C03645=1176.042,92.652,-51.203,-179.040,6.178,148.830
C03646=1176.047,92.403,-51.185,-179.044,6.176,148.831
C03647=1176.052,92.154,-51.167,-179.046,6.175,148.831
C03648=1176.057,91.904,-51.149,-179.048,6.174,148.832
C03649=1176.062,91.655,-51.131,-179.051,6.173,148.832
C03650=1176.066,91.406,-51.113,-179.054,6.172,148.833
C03651=1176.071,91.156,-51.095,-179.056,6.171,148.833
C03652=1176.076,90.906,-51.077,-179.059,6.169,148.834
C03653=1176.081,90.657,-51.059,-179.061,6.168,148.834
C03654=1176.086,90.408,-51.042,-179.064,6.167,148.835
C03655=1176.091,90.159,-51.024,-179.067,6.166,148.835
C03656=1176.096,89.910,-51.006,-179.070,6.165,148.836
C03657=1176.101,89.660,-50.988,-179.073,6.163,148.836
C03658=1176.106,89.411,-50.970,-179.075,6.162,148.837
C03659=1176.111,89.162,-50.952,-179.078,6.161,148.837
C03660=1176.116,88.912,-50.934,-179.080,6.160,148.838
C03661=1176.120,88.664,-50.917,-179.083,6.159,148.839
C03662=1176.125,88.414,-50.900,-179.085,6.158,148.839
C03663=1176.130,88.165,-50.882,-179.089,6.156,148.840
C03664=1176.135,87.915,-50.864,-179.091,6.155,148.840
C03665=1176.140,87.666,-50.846,-179.093,6.154,148.840
C03666=1176.145,87.416,-50.828,-179.096,6.153,148.841
C03667=1176.150,87.167,-50.811,-179.099,6.151,148.842
C03668=1176.155,86.918,-50.793,-179.101,6.151,148.842
C03669=1176.159,86.669,-50.776,-179.104,6.149,148.843
C03670=1176.164,86.419,-50.758,-179.106,6.148,148.843
C03671=1176.169,86.170,-50.740,-179.109,6.147,148.844
C03672=1176.174,85.920,-50.723,-179.112,6.146,148.844
C03673=1176.179,85.671,-50.705,-179.115,6.145,148.845
C03674=1176.184,85.422,-50.687,-179.117,6.144,148.845
C03675=1176.189,85.173,-50.670,-179.120,6.142,148.846
C03676=1176.193,84.923,-50.652,-179.122,6.142,148.846
C03677=1176.198,84.674,-50.634,-179.125,6.140,148.847
C03678=1176.204,84.424,-50.617,-179.128,6.139,148.847
C03679=1176.209,84.175,-50.599,-179.130,6.138,148.848
C03680=1176.213,83.926,-50.582,-179.133,6.137,148.848
C03681=1176.218,83.677,-50.564,-179.136,6.135,148.849
C03682=1176.223,83.427,-50.547,-179.138,6.135,148.849
C03683=1176.228,83.178,-50.529,-179.141,6.133,148.850
C03684=1176.232,82.929,-50.512,-179.144,6.133,148.851
C03685=1176.237,82.679,-50.494,-179.146,6.131,148.851
C03686=1176.242,82.430,-50.476,-179.149,6.130,148.852
C03687=1176.248,82.180,-50.459,-179.152,6.129,148.852
C03688=1176.252,81.931,-50.442,-179.154,6.128,148.852
C03689=1176.257,81.681,-50.424,-179.157,6.126,148.853
C03690=1176.262,81.432,-50.406,-179.159,6.125,148.854
C03691=1176.267,81.183,-50.390,-179.162,6.124,148.854
C03692=1176.272,80.934,-50.372,-179.165,6.123,148.855
C03693=1176.277,80.665,-50.353,-179.168,6.122,148.855
C03694=1176.283,80.397,-50.335,-179.170,6.121,148.856
C03695=1176.288,80.129,-50.316,-179.173,6.120,148.856
C03696=1176.293,79.860,-50.298,-179.176,6.118,148.857
C03697=1176.298,79.611,-50.280,-179.179,6.117,148.857
C03698=1176.303,79.361,-50.262,-179.182,6.116,148.858
C03699=1176.308,79.112,-50.246,-179.184,6.115,148.858
C03700=1176.312,78.863,-50.228,-179.187,6.114,148.859
C03701=1176.317,78.613,-50.211,-179.189,6.113,148.860
C03702=1176.323,78.364,-50.194,-179.192,6.112,148.860
C03703=1176.328,78.115,-50.176,-179.195,6.111,148.861
C03704=1176.332,77.866,-50.159,-179.197,6.110,148.861
C03705=1176.337,77.616,-50.142,-179.200,6.108,148.862
C03706=1176.342,77.367,-50.124,-179.202,6.108,148.862
C03707=1176.347,77.117,-50.108,-179.205,6.106,148.863
C03708=1176.353,76.868,-50.091,-179.207,6.105,148.863
C03709=1176.357,76.619,-50.073,-179.211,6.104,148.864
C03710=1176.362,76.369,-50.056,-179.213,6.103,148.864
C03711=1176.366,76.120,-50.039,-179.216,6.102,148.865
C03712=1176.372,75.870,-50.022,-179.218,6.101,148.865
C03713=1176.377,75.621,-50.004,-179.221,6.100,148.866
C03714=1176.382,75.372,-49.988,-179.223,6.099,148.866
C03715=1176.387,75.122,-49.971,-179.226,6.098,148.867
C03716=1176.391,74.873,-49.954,-179.229,6.096,148.868
C03717=1176.396,74.624,-49.936,-179.231,6.096,148.868
C03718=1176.401,74.374,-49.919,-179.234,6.094,148.869
C03719=1176.407,74.125,-49.902,-179.237,6.094,148.869
C03720=1176.411,73.876,-49.886,-179.239,6.093,148.870
C03721=1176.416,73.626,-49.868,-179.242,6.091,148.870
C03722=1176.420,73.377,-49.851,-179.244,6.091,148.871
C03723=1176.426,73.127,-49.834,-179.248,6.089,148.871
C03724=1176.431,72.878,-49.817,-179.250,6.088,148.872
C03725=1176.436,72.629,-49.800,-179.253,6.087,148.873
C03726=1176.440,72.379,-49.783,-179.255,6.086,148.873
C03727=1176.446,72.129,-49.766,-179.258,6.086,148.874
C03728=1176.451,71.880,-49.750,-179.260,6.084,148.874
C03729=1176.455,71.632,-49.733,-179.263,6.083,148.875
C03730=1176.460,71.382,-49.715,-179.266,6.082,148.875
C03731=1176.465,71.132,-49.699,-179.268,6.081,148.876
C03732=1176.470,70.883,-49.682,-179.271,6.080,148.876
C03733=1176.475,70.634,-49.665,-179.273,6.079,148.877
C03734=1176.480,70.384,-49.648,-179.276,6.078,148.877
C03735=1176.485,70.135,-49.631,-179.279,6.076,148.878
C03736=1176.490,69.886,-49.615,-179.281,6.076,148.878
C03737=1176.495,69.636,-49.598,-179.284,6.074,148.879
C03738=1176.499,69.386,-49.581,-179.287,6.074,148.880
C03739=1176.505,69.137,-49.564,-179.289,6.073,148.880
C03740=1176.510,68.888,-49.547,-179.292,6.071,148.881
C03741=1176.514,68.638,-49.531,-179.294,6.070,148.881
C03742=1176.520,68.389,-49.514,-179.297,6.069,148.882
C03743=1176.524,68.140,-49.497,-179.300,6.069,148.882
C03744=1176.529,67.890,-49.480,-179.302,6.068,148.883
C03745=1176.535,67.641,-49.463,-179.305,6.066,148.883
C03746=1176.539,67.392,-49.447,-179.307,6.066,148.884
C03747=1176.544,67.142,-49.430,-179.310,6.065,148.885
C03748=1176.549,66.892,-49.413,-179.313,6.063,148.885
C03749=1176.554,66.644,-49.397,-179.315,6.063,148.886
C03750=1176.559,66.394,-49.380,-179.318,6.061,148.886
C03751=1176.564,66.145,-49.363,-179.321,6.061,148.887
C03752=1176.569,65.896,-49.346,-179.323,6.060,148.887
C03753=1176.574,65.645,-49.330,-179.326,6.058,148.888
C03754=1176.579,65.397,-49.314,-179.328,6.057,148.888
C03755=1176.584,65.147,-49.297,-179.331,6.057,148.889
C03756=1176.588,64.897,-49.280,-179.334,6.055,148.889
C03757=1176.593,64.649,-49.264,-179.336,6.055,148.890
C03758=1176.599,64.399,-49.247,-179.339,6.053,148.890
C03759=1176.603,64.149,-49.230,-179.342,6.053,148.891
C03760=1176.609,63.900,-49.214,-179.344,6.052,148.892
C03761=1176.613,63.650,-49.198,-179.347,6.050,148.892
C03762=1176.619,63.401,-49.181,-179.349,6.049,148.893
C03763=1176.623,63.152,-49.164,-179.352,6.049,148.893
C03764=1176.628,62.902,-49.147,-179.355,6.047,148.894
C03765=1176.633,62.653,-49.132,-179.357,6.047,148.894
C03766=1176.638,62.404,-49.115,-179.359,6.046,148.895
C03767=1176.644,62.154,-49.098,-179.363,6.045,148.895
C03768=1176.648,61.905,-49.082,-179.365,6.044,148.896
C03769=1176.653,61.655,-49.066,-179.368,6.042,148.897
C03770=1176.658,61.406,-49.049,-179.371,6.042,148.897
C03771=1176.662,61.157,-49.033,-179.373,6.041,148.898
C03772=1176.668,60.907,-49.017,-179.376,6.040,148.898
C03773=1176.673,60.657,-49.000,-179.378,6.039,148.899
C03774=1176.678,60.409,-48.984,-179.381,6.038,148.899
C03775=1176.683,60.158,-48.968,-179.383,6.036,148.900
C03776=1176.688,59.910,-48.951,-179.386,6.036,148.901
C03777=1176.692,59.660,-48.935,-179.388,6.035,148.901
C03778=1176.697,59.410,-48.919,-179.391,6.034,148.902
C03779=1176.702,59.161,-48.902,-179.394,6.033,148.902
C03780=1176.707,58.912,-48.885,-179.396,6.032,148.903
C03781=1176.713,58.662,-48.869,-179.399,6.031,148.903
C03782=1176.717,58.413,-48.853,-179.402,6.030,148.904
C03783=1176.722,58.164,-48.837,-179.404,6.030,148.905
C03784=1176.727,57.914,-48.821,-179.407,6.028,148.905
C03785=1176.732,57.665,-48.804,-179.410,6.027,148.906
C03786=1176.737,57.415,-48.788,-179.412,6.027,148.906
C03787=1176.742,57.166,-48.772,-179.415,6.025,148.907
C03788=1176.747,56.916,-48.756,-179.417,6.024,148.907
C03789=1176.752,56.667,-48.740,-179.420,6.024,148.908
C03790=1176.756,56.418,-48.723,-179.423,6.022,148.908
C03791=1176.762,56.168,-48.707,-179.425,6.022,148.909
C03792=1176.767,55.919,-48.690,-179.427,6.021,148.909
C03793=1176.772,55.669,-48.675,-179.431,6.019,148.910
C03794=1176.777,55.420,-48.658,-179.433,6.019,148.911
C03795=1176.782,55.170,-48.642,-179.435,6.018,148.911
C03796=1176.787,54.921,-48.626,-179.438,6.018,148.912
C03797=1176.792,54.652,-48.609,-179.441,6.016,148.912
C03798=1176.798,54.384,-48.592,-179.443,6.015,148.913
C03799=1176.803,54.115,-48.575,-179.447,6.014,148.914
C03800=1176.808,53.846,-48.557,-179.449,6.014,148.914
C03801=1176.814,53.597,-48.541,-179.452,6.012,148.915
C03802=1176.819,53.348,-48.525,-179.455,6.011,148.915
C03803=1176.823,53.098,-48.509,-179.457,6.010,148.916
C03804=1176.829,52.849,-48.493,-179.460,6.009,148.916
C03805=1176.833,52.600,-48.476,-179.462,6.008,148.917
C03806=1176.839,52.350,-48.461,-179.465,6.008,148.918
C03807=1176.843,52.100,-48.445,-179.468,6.006,148.918
C03808=1176.849,51.851,-48.429,-179.470,6.006,148.919
C03809=1176.853,51.602,-48.414,-179.473,6.005,148.919
C03810=1176.858,51.352,-48.398,-179.475,6.004,148.920
C03811=1176.863,51.103,-48.381,-179.478,6.003,148.920
C03812=1176.868,50.853,-48.365,-179.480,6.002,148.921
C03813=1176.873,50.604,-48.350,-179.483,6.001,148.922
C03814=1176.878,50.355,-48.334,-179.486,6.000,148.922
C03815=1176.883,50.105,-48.318,-179.488,5.999,148.923
C03816=1176.888,49.856,-48.302,-179.491,5.999,148.923
C03817=1176.894,49.607,-48.286,-179.493,5.998,148.924
C03818=1176.898,49.357,-48.270,-179.496,5.997,148.924
C03819=1176.903,49.108,-48.255,-179.498,5.996,148.925
C03820=1176.908,48.857,-48.239,-179.501,5.995,148.926
C03821=1176.913,48.609,-48.222,-179.504,5.995,148.926
C03822=1176.918,48.359,-48.207,-179.506,5.993,148.927
C03823=1176.923,48.109,-48.191,-179.509,5.993,148.927
C03824=1176.928,47.860,-48.175,-179.511,5.992,148.928
C03825=1176.933,47.611,-48.160,-179.515,5.990,148.928
C03826=1176.938,47.361,-48.144,-179.517,5.989,148.929
C03827=1176.943,47.112,-48.128,-179.519,5.989,148.930
C03828=1176.948,46.862,-48.112,-179.522,5.988,148.930
C03829=1176.953,46.612,-48.097,-179.525,5.987,148.931
C03830=1176.957,46.364,-48.081,-179.527,5.986,148.931
C03831=1176.963,46.114,-48.065,-179.529,5.985,148.932
C03832=1176.968,45.864,-48.049,-179.532,5.985,148.932
C03833=1176.973,45.615,-48.034,-179.535,5.984,148.933
C03834=1176.978,45.366,-48.019,-179.537,5.983,148.934
C03835=1176.982,45.116,-48.003,-179.540,5.982,148.934
C03836=1176.988,44.866,-47.987,-179.542,5.981,148.935
C03837=1176.993,44.618,-47.971,-179.546,5.980,148.935
C03838=1176.998,44.368,-47.955,-179.548,5.979,148.936
C03839=1177.002,44.118,-47.940,-179.550,5.979,148.936
C03840=1177.008,43.869,-47.924,-179.553,5.978,148.937
C03841=1177.013,43.619,-47.909,-179.556,5.976,148.938
C03842=1177.017,43.370,-47.893,-179.558,5.976,148.938
C03843=1177.023,43.120,-47.878,-179.560,5.975,148.939
C03844=1177.028,42.871,-47.862,-179.563,5.975,148.939
C03845=1177.033,42.621,-47.847,-179.566,5.973,148.940
C03846=1177.037,42.372,-47.831,-179.569,5.972,148.940
C03847=1177.043,42.122,-47.816,-179.571,5.972,148.941
C03848=1177.048,41.873,-47.800,-179.573,5.971,148.942
C03849=1177.053,41.624,-47.785,-179.576,5.971,148.942
C03850=1177.058,41.374,-47.769,-179.579,5.969,148.943
C03851=1177.063,41.124,-47.754,-179.581,5.968,148.943
C03852=1177.068,40.875,-47.739,-179.584,5.968,148.944
C03853=1177.073,40.626,-47.723,-179.586,5.967,148.945
C03854=1177.078,40.376,-47.707,-179.589,5.966,148.945
C03855=1177.082,40.127,-47.692,-179.592,5.965,148.946
C03856=1177.088,39.877,-47.676,-179.594,5.964,148.946
C03857=1177.093,39.628,-47.661,-179.597,5.964,148.947
C03858=1177.098,39.379,-47.646,-179.599,5.963,148.947
C03859=1177.103,39.129,-47.630,-179.602,5.962,148.948
C03860=1177.107,38.880,-47.615,-179.605,5.961,148.949
C03861=1177.113,38.629,-47.600,-179.607,5.960,148.949
C03862=1177.118,38.380,-47.584,-179.610,5.960,148.950
C03863=1177.123,38.131,-47.569,-179.612,5.958,148.950
C03864=1177.128,37.882,-47.554,-179.615,5.958,148.951
C03865=1177.132,37.632,-47.539,-179.618,5.957,148.952
C03866=1177.138,37.382,-47.523,-179.620,5.956,148.952
C03867=1177.143,37.133,-47.507,-179.622,5.956,148.953
C03868=1177.148,36.883,-47.493,-179.625,5.954,148.953
C03869=1177.154,36.634,-47.477,-179.628,5.954,148.954
C03870=1177.158,36.385,-47.462,-179.630,5.953,148.955
C03871=1177.164,36.135,-47.447,-179.633,5.952,148.955
C03872=1177.168,35.886,-47.432,-179.635,5.952,148.956
C03873=1177.173,35.636,-47.417,-179.638,5.950,148.956
C03874=1177.178,35.386,-47.402,-179.641,5.950,148.957
C03875=1177.183,35.137,-47.386,-179.643,5.949,148.958
C03876=1177.188,34.888,-47.371,-179.645,5.948,148.958
C03877=1177.193,34.639,-47.356,-179.648,5.948,148.959
C03878=1177.198,34.389,-47.341,-179.651,5.946,148.959
C03879=1177.204,34.139,-47.326,-179.653,5.946,148.960
C03880=1177.208,33.890,-47.310,-179.656,5.945,148.960
C03881=1177.213,33.640,-47.295,-179.658,5.944,148.961
C03882=1177.218,33.391,-47.280,-179.661,5.944,148.962
C03883=1177.224,33.141,-47.265,-179.664,5.943,148.962
C03884=1177.228,32.892,-47.250,-179.666,5.942,148.963
C03885=1177.234,32.642,-47.235,-179.669,5.941,148.963
C03886=1177.239,32.393,-47.220,-179.671,5.940,148.964
C03887=1177.244,32.144,-47.204,-179.674,5.940,148.964
C03888=1177.249,31.894,-47.190,-179.676,5.939,148.965
C03889=1177.254,31.645,-47.175,-179.679,5.938,148.966
C03890=1177.259,31.394,-47.160,-179.682,5.937,148.966
C03891=1177.263,31.145,-47.145,-179.684,5.937,148.967
C03892=1177.269,30.896,-47.129,-179.687,5.936,148.967
C03893=1177.274,30.646,-47.115,-179.689,5.935,148.968
C03894=1177.278,30.397,-47.100,-179.691,5.934,148.969
C03895=1177.284,30.147,-47.084,-179.695,5.933,148.969
C03896=1177.289,29.898,-47.070,-179.697,5.933,148.970
C03897=1177.294,29.648,-47.055,-179.699,5.932,148.970
C03898=1177.299,29.399,-47.040,-179.702,5.931,148.971
C03899=1177.304,29.149,-47.025,-179.705,5.931,148.972
C03900=1177.309,28.899,-47.010,-179.707,5.930,148.972
C03901=1177.314,28.631,-46.995,-179.710,5.929,148.973
C03902=1177.320,28.362,-46.978,-179.713,5.928,148.973
C03903=1177.325,28.093,-46.962,-179.715,5.928,148.974
C03904=1177.330,27.825,-46.946,-179.718,5.926,148.975
C03905=1177.336,27.575,-46.931,-179.721,5.925,148.975
C03906=1177.341,27.325,-46.916,-179.723,5.925,148.976
C03907=1177.345,27.076,-46.902,-179.726,5.924,148.976
C03908=1177.351,26.826,-46.887,-179.728,5.924,148.977
C03909=1177.356,26.577,-46.872,-179.731,5.923,148.978
C03910=1177.360,26.328,-46.857,-179.733,5.922,148.978
C03911=1177.366,26.078,-46.842,-179.736,5.921,148.979
C03912=1177.371,25.828,-46.827,-179.739,5.920,148.980
C03913=1177.376,25.579,-46.813,-179.741,5.920,148.980
C03914=1177.381,25.329,-46.799,-179.744,5.919,148.981
C03915=1177.386,25.080,-46.783,-179.746,5.918,148.981
C03916=1177.391,24.830,-46.769,-179.749,5.918,148.982
C03917=1177.396,24.581,-46.754,-179.751,5.917,148.983
C03918=1177.401,24.331,-46.740,-179.754,5.916,148.983
C03919=1177.406,24.081,-46.725,-179.757,5.915,148.984
C03920=1177.411,23.832,-46.710,-179.759,5.915,148.984
C03921=1177.416,23.582,-46.696,-179.761,5.914,148.985
C03922=1177.421,23.334,-46.681,-179.764,5.913,148.985
C03923=1177.427,23.084,-46.666,-179.767,5.913,148.986
C03924=1177.432,22.834,-46.652,-179.769,5.912,148.987
C03925=1177.437,22.585,-46.637,-179.772,5.911,148.987
C03926=1177.441,22.335,-46.623,-179.774,5.910,148.988
C03927=1177.446,22.086,-46.608,-179.777,5.909,148.988
C03928=1177.452,21.836,-46.593,-179.780,5.909,148.989
C03929=1177.457,21.587,-46.578,-179.782,5.908,148.990
C03930=1177.462,21.337,-46.564,-179.784,5.907,148.990
C03931=1177.467,21.087,-46.550,-179.787,5.907,148.991
C03932=1177.471,20.838,-46.535,-179.789,5.906,148.991
C03933=1177.476,20.588,-46.521,-179.792,5.906,148.992
C03934=1177.483,20.339,-46.506,-179.795,5.905,148.993
C03935=1177.488,20.089,-46.492,-179.797,5.903,148.993
C03936=1177.492,19.840,-46.477,-179.800,5.903,148.994
C03937=1177.497,19.590,-46.463,-179.803,5.903,148.995
C03938=1177.502,19.341,-46.448,-179.805,5.902,148.995
C03939=1177.507,19.091,-46.434,-179.807,5.901,148.996
C03940=1177.512,18.841,-46.420,-179.810,5.900,148.996
C03941=1177.517,18.592,-46.405,-179.812,5.900,148.997
C03942=1177.523,18.343,-46.390,-179.815,5.899,148.998
C03943=1177.528,18.093,-46.376,-179.817,5.899,148.998
C03944=1177.533,17.843,-46.362,-179.820,5.898,148.999
C03945=1177.538,17.594,-46.347,-179.823,5.897,148.999
C03946=1177.543,17.344,-46.333,-179.825,5.896,149.000
C03947=1177.547,17.095,-46.318,-179.828,5.895,149.000
C03948=1177.552,16.845,-46.304,-179.830,5.895,149.001
C03949=1177.558,16.596,-46.290,-179.833,5.894,149.002
C03950=1177.563,16.347,-46.276,-179.835,5.894,149.002
C03951=1177.568,16.097,-46.261,-179.838,5.893,149.003
C03952=1177.573,15.847,-46.247,-179.840,5.892,149.003
C03953=1177.578,15.597,-46.233,-179.843,5.892,149.004
C03954=1177.583,15.348,-46.219,-179.845,5.891,149.005
C03955=1177.588,15.099,-46.205,-179.847,5.890,149.005
C03956=1177.593,14.849,-46.190,-179.850,5.890,149.006
C03957=1177.598,14.600,-46.175,-179.853,5.889,149.007
C03958=1177.603,14.350,-46.161,-179.855,5.888,149.007
C03959=1177.608,14.100,-46.147,-179.858,5.887,149.008
C03960=1177.613,13.851,-46.133,-179.860,5.887,149.008
C03961=1177.618,13.602,-46.119,-179.863,5.886,149.009
C03962=1177.623,13.352,-46.104,-179.866,5.886,149.010
C03963=1177.628,13.102,-46.090,-179.868,5.885,149.010
C03964=1177.634,12.853,-46.076,-179.870,5.884,149.011
C03965=1177.639,12.604,-46.062,-179.873,5.884,149.011
C03966=1177.644,12.354,-46.048,-179.875,5.883,149.012
C03967=1177.649,12.104,-46.033,-179.878,5.882,149.013
C03968=1177.654,11.855,-46.019,-179.881,5.882,149.013
C03969=1177.659,11.605,-46.005,-179.883,5.881,149.014
C03970=1177.664,11.355,-45.992,-179.885,5.881,149.014
C03971=1177.669,11.105,-45.977,-179.888,5.880,149.015
C03972=1177.675,10.856,-45.963,-179.891,5.878,149.016
C03973=1177.680,10.607,-45.949,-179.893,5.878,149.016
C03974=1177.685,10.357,-45.935,-179.896,5.878,149.017
C03975=1177.690,10.107,-45.921,-179.898,5.877,149.017
C03976=1177.695,9.858,-45.907,-179.901,5.876,149.018
C03977=1177.700,9.609,-45.893,-179.904,5.876,149.019
C03978=1177.704,9.359,-45.879,-179.906,5.875,149.019
C03979=1177.709,9.109,-45.864,-179.908,5.874,149.020
C03980=1177.715,8.860,-45.851,-179.911,5.874,149.021
C03981=1177.720,8.610,-45.837,-179.913,5.873,149.021
C03982=1177.725,8.360,-45.823,-179.916,5.873,149.022
C03983=1177.731,8.111,-45.809,-179.918,5.872,149.022
C03984=1177.735,7.862,-45.795,-179.921,5.871,149.023
C03985=1177.740,7.612,-45.781,-179.923,5.871,149.024
C03986=1177.746,7.363,-45.768,-179.926,5.870,149.024
C03987=1177.751,7.113,-45.753,-179.928,5.870,149.025
C03988=1177.756,6.863,-45.739,-179.931,5.869,149.025
C03989=1177.761,6.614,-45.725,-179.933,5.869,149.026
C03990=1177.765,6.365,-45.711,-179.936,5.868,149.026
C03991=1177.771,6.115,-45.698,-179.938,5.867,149.027
C03992=1177.776,5.865,-45.684,-179.941,5.867,149.028
C03993=1177.781,5.616,-45.670,-179.943,5.866,149.028
C03994=1177.786,5.366,-45.655,-179.946,5.865,149.029
C03995=1177.791,5.116,-45.642,-179.948,5.865,149.030
C03996=1177.796,4.867,-45.629,-179.951,5.864,149.030
C03997=1177.801,4.617,-45.614,-179.953,5.864,149.031
C03998=1177.807,4.368,-45.600,-179.956,5.862,149.032
C03999=1177.812,4.118,-45.587,-179.959,5.862,149.032
C04000=1177.816,3.869,-45.573,-179.961,5.861,149.033
C04001=1177.822,3.620,-45.559,-179.964,5.861,149.033
C04002=1177.827,3.369,-45.546,-179.966,5.860,149.034
C04003=1177.832,3.120,-45.531,-179.969,5.859,149.035
C04004=1177.837,2.871,-45.518,-179.971,5.859,149.035
C04005=1177.842,2.601,-45.503,-179.974,5.858,149.036
C04006=1177.848,2.332,-45.488,-179.976,5.858,149.036
C04007=1177.853,2.063,-45.473,-179.979,5.857,149.037
C04008=1177.860,1.793,-45.459,-179.982,5.857,149.038
C04009=1177.864,1.544,-45.445,-179.984,5.856,149.038
C04010=1177.869,1.295,-45.432,-179.987,5.856,149.039
C04011=1177.875,1.045,-45.418,-179.989,5.855,149.040
C04012=1177.879,0.795,-45.404,-179.992,5.854,149.040
C04013=1177.885,0.546,-45.391,-179.994,5.854,149.041
C04014=1177.890,0.296,-45.377,-179.996,5.853,149.041
C04015=1177.895,0.047,-45.363,-179.999,5.853,149.042
C04016=1177.900,-0.203,-45.350,179.998,5.852,149.043
C04017=1177.905,-0.453,-45.336,179.996,5.851,149.043
C04018=1177.910,-0.703,-45.322,179.993,5.851,149.044
C04019=1177.915,-0.952,-45.309,179.991,5.850,149.045
C04020=1177.921,-1.202,-45.296,179.989,5.849,149.045
C04021=1177.926,-1.451,-45.281,179.986,5.849,149.046
C04022=1177.931,-1.701,-45.269,179.983,5.849,149.046
C04023=1177.936,-1.950,-45.254,179.981,5.848,149.047
C04024=1177.941,-2.200,-45.242,179.978,5.847,149.048
C04025=1177.946,-2.449,-45.228,179.976,5.847,149.048
C04026=1177.952,-2.699,-45.214,179.974,5.846,149.049
C04027=1177.956,-2.948,-45.201,179.971,5.845,149.049
C04028=1177.962,-3.198,-45.187,179.968,5.845,149.050
C04029=1177.966,-3.447,-45.174,179.966,5.844,149.051
C04030=1177.971,-3.698,-45.160,179.963,5.844,149.051
C04031=1177.977,-3.947,-45.146,179.961,5.843,149.052
C04032=1177.981,-4.197,-45.133,179.959,5.842,149.052
C04033=1177.987,-4.446,-45.120,179.956,5.842,149.053
C04034=1177.991,-4.696,-45.106,179.953,5.841,149.054
C04035=1177.997,-4.945,-45.093,179.951,5.841,149.054
C04036=1178.001,-5.195,-45.080,179.949,5.840,149.055
C04037=1178.007,-5.444,-45.066,179.946,5.840,149.056
C04038=1178.012,-5.694,-45.054,179.944,5.839,149.056
C04039=1178.017,-5.943,-45.040,179.941,5.838,149.057
C04040=1178.022,-6.193,-45.027,179.938,5.838,149.058
C04041=1178.028,-6.443,-45.013,179.936,5.837,149.058
C04042=1178.033,-6.692,-44.999,179.934,5.837,149.059
C04043=1178.038,-6.942,-44.986,179.931,5.836,149.059
C04044=1178.043,-7.191,-44.973,179.929,5.835,149.060
C04045=1178.048,-7.441,-44.960,179.926,5.835,149.061
C04046=1178.053,-7.691,-44.947,179.923,5.834,149.061
C04047=1178.058,-7.941,-44.933,179.921,5.834,149.062
C04048=1178.063,-8.190,-44.920,179.919,5.834,149.062
C04049=1178.068,-8.440,-44.907,179.917,5.833,149.063
C04050=1178.073,-8.689,-44.894,179.914,5.833,149.064
C04051=1178.079,-8.938,-44.880,179.912,5.832,149.064
C04052=1178.083,-9.188,-44.867,179.909,5.832,149.065
C04053=1178.089,-9.438,-44.854,179.906,5.831,149.066
C04054=1178.094,-9.688,-44.841,179.904,5.830,149.066
C04055=1178.099,-9.937,-44.827,179.902,5.830,149.067
C04056=1178.104,-10.187,-44.814,179.899,5.830,149.067
C04057=1178.109,-10.436,-44.801,179.897,5.829,149.068
C04058=1178.115,-10.686,-44.788,179.894,5.828,149.069
C04059=1178.119,-10.935,-44.775,179.891,5.828,149.069
C04060=1178.125,-11.185,-44.761,179.889,5.827,149.070
C04061=1178.130,-11.435,-44.748,179.887,5.826,149.070
C04062=1178.135,-11.684,-44.736,179.884,5.826,149.071
C04063=1178.140,-11.934,-44.723,179.882,5.825,149.072
C04064=1178.145,-12.184,-44.710,179.879,5.825,149.072
C04065=1178.151,-12.433,-44.696,179.877,5.825,149.073
C04066=1178.155,-12.683,-44.683,179.875,5.824,149.073
C04067=1178.160,-12.932,-44.670,179.872,5.824,149.074
C04068=1178.166,-13.182,-44.657,179.870,5.823,149.075
C04069=1178.171,-13.432,-44.644,179.867,5.822,149.075
C04070=1178.176,-13.681,-44.631,179.865,5.822,149.076
C04071=1178.182,-13.931,-44.618,179.862,5.822,149.077
C04072=1178.186,-14.180,-44.605,179.860,5.821,149.077
C04073=1178.191,-14.429,-44.592,179.857,5.820,149.078
C04074=1178.196,-14.680,-44.578,179.855,5.820,149.079
C04075=1178.201,-14.929,-44.566,179.852,5.819,149.079
C04076=1178.206,-15.178,-44.553,179.850,5.819,149.080
C04077=1178.212,-15.429,-44.540,179.847,5.818,149.080
C04078=1178.217,-15.678,-44.527,179.844,5.818,149.081
C04079=1178.222,-15.927,-44.514,179.843,5.818,149.082
C04080=1178.227,-16.178,-44.501,179.840,5.817,149.082
C04081=1178.232,-16.427,-44.488,179.837,5.817,149.083
C04082=1178.237,-16.676,-44.476,179.835,5.816,149.083
C04083=1178.243,-16.926,-44.463,179.833,5.815,149.084
C04084=1178.248,-17.176,-44.449,179.830,5.815,149.085
C04085=1178.253,-17.425,-44.437,179.828,5.814,149.085
C04086=1178.258,-17.675,-44.424,179.825,5.814,149.086
C04087=1178.263,-17.925,-44.411,179.822,5.813,149.087
C04088=1178.268,-18.174,-44.398,179.820,5.812,149.087
C04089=1178.274,-18.424,-44.386,179.818,5.812,149.088
C04090=1178.278,-18.674,-44.373,179.816,5.812,149.089
C04091=1178.284,-18.923,-44.359,179.813,5.811,149.089
C04092=1178.289,-19.173,-44.347,179.811,5.811,149.090
C04093=1178.294,-19.422,-44.334,179.808,5.811,149.090
C04094=1178.299,-19.672,-44.321,179.806,5.810,149.091
C04095=1178.304,-19.921,-44.309,179.803,5.809,149.092
C04096=1178.310,-20.171,-44.295,179.801,5.809,149.092
C04097=1178.315,-20.420,-44.283,179.798,5.808,149.093
C04098=1178.320,-20.671,-44.271,179.796,5.808,149.093
C04099=1178.325,-20.920,-44.258,179.794,5.808,149.094
C04100=1178.330,-21.169,-44.245,179.791,5.807,149.095
C04101=1178.336,-21.419,-44.232,179.789,5.807,149.095
C04102=1178.340,-21.669,-44.219,179.786,5.806,149.096
C04103=1178.345,-21.918,-44.207,179.784,5.806,149.097
C04104=1178.351,-22.168,-44.194,179.781,5.805,149.097
C04105=1178.356,-22.417,-44.181,179.779,5.804,149.098
C04106=1178.361,-22.668,-44.169,179.776,5.804,149.099
C04107=1178.366,-22.917,-44.156,179.774,5.803,149.099
C04108=1178.372,-23.167,-44.143,179.772,5.804,149.100
C04109=1178.377,-23.436,-44.130,179.769,5.803,149.100
C04110=1178.383,-23.706,-44.116,179.766,5.803,149.101
C04111=1178.388,-23.976,-44.103,179.763,5.801,149.102
C04112=1178.393,-24.246,-44.089,179.761,5.801,149.102
C04113=1178.398,-24.495,-44.076,179.759,5.801,149.103
C04114=1178.404,-24.745,-44.063,179.756,5.800,149.104
C04115=1178.410,-24.995,-44.051,179.754,5.800,149.104
C04116=1178.415,-25.244,-44.039,179.751,5.799,149.105
C04117=1178.419,-25.494,-44.026,179.749,5.799,149.105
C04118=1178.424,-25.743,-44.013,179.746,5.798,149.106
C04119=1178.430,-25.993,-44.001,179.744,5.797,149.107
C04120=1178.435,-26.243,-43.989,179.742,5.798,149.107
C04121=1178.440,-26.492,-43.976,179.739,5.797,149.108
C04122=1178.445,-26.742,-43.963,179.737,5.797,149.109
C04123=1178.450,-26.992,-43.951,179.734,5.796,149.109
C04124=1178.455,-27.241,-43.939,179.732,5.796,149.110
C04125=1178.460,-27.491,-43.926,179.730,5.795,149.110
C04126=1178.466,-27.740,-43.914,179.727,5.794,149.111
C04127=1178.471,-27.990,-43.902,179.724,5.794,149.112
C04128=1178.475,-28.240,-43.889,179.723,5.794,149.112
C04129=1178.481,-28.490,-43.877,179.720,5.793,149.113
C04130=1178.486,-28.739,-43.864,179.717,5.793,149.114
C04131=1178.491,-28.988,-43.852,179.715,5.792,149.114
C04132=1178.496,-29.238,-43.840,179.712,5.792,149.115
C04133=1178.502,-29.488,-43.827,179.710,5.791,149.116
C04134=1178.507,-29.738,-43.815,179.708,5.792,149.116
C04135=1178.512,-29.987,-43.803,179.706,5.791,149.117
C04136=1178.517,-30.237,-43.790,179.703,5.790,149.117
C04137=1178.522,-30.487,-43.778,179.700,5.790,149.118
C04138=1178.527,-30.736,-43.765,179.698,5.789,149.119
C04139=1178.533,-30.986,-43.753,179.695,5.789,149.119
C04140=1178.538,-31.235,-43.741,179.693,5.788,149.120
C04141=1178.543,-31.485,-43.728,179.691,5.788,149.120
C04142=1178.548,-31.735,-43.716,179.688,5.788,149.121
C04143=1178.553,-31.984,-43.704,179.686,5.787,149.122
C04144=1178.559,-32.234,-43.692,179.684,5.787,149.122
C04145=1178.564,-32.483,-43.679,179.681,5.786,149.123
C04146=1178.569,-32.734,-43.667,179.678,5.786,149.124
C04147=1178.574,-32.983,-43.654,179.677,5.786,149.124
C04148=1178.579,-33.233,-43.642,179.674,5.785,149.125
C04149=1178.584,-33.482,-43.630,179.671,5.785,149.126
C04150=1178.589,-33.732,-43.618,179.669,5.784,149.126
C04151=1178.594,-33.981,-43.606,179.667,5.784,149.127
C04152=1178.600,-34.231,-43.594,179.664,5.783,149.127
C04153=1178.605,-34.481,-43.581,179.662,5.783,149.128
C04154=1178.610,-34.731,-43.569,179.660,5.783,149.129
C04155=1178.615,-34.980,-43.557,179.657,5.782,149.129
C04156=1178.621,-35.230,-43.545,179.655,5.781,149.130
C04157=1178.626,-35.480,-43.533,179.652,5.781,149.130
C04158=1178.631,-35.729,-43.520,179.650,5.781,149.131
C04159=1178.636,-35.979,-43.509,179.648,5.780,149.132
C04160=1178.641,-36.228,-43.497,179.645,5.780,149.132
C04161=1178.647,-36.478,-43.485,179.643,5.780,149.133
C04162=1178.652,-36.728,-43.473,179.640,5.779,149.133
C04163=1178.657,-36.977,-43.460,179.638,5.778,149.134
C04164=1178.663,-37.227,-43.448,179.636,5.779,149.135
C04165=1178.667,-37.476,-43.436,179.633,5.778,149.135
C04166=1178.672,-37.726,-43.424,179.631,5.777,149.136
C04167=1178.678,-37.976,-43.413,179.628,5.777,149.137
C04168=1178.683,-38.225,-43.400,179.626,5.776,149.137
C04169=1178.688,-38.475,-43.388,179.624,5.777,149.138
C04170=1178.694,-38.725,-43.376,179.621,5.776,149.139
C04171=1178.698,-38.974,-43.364,179.619,5.776,149.139
C04172=1178.704,-39.224,-43.352,179.616,5.775,149.140
C04173=1178.709,-39.474,-43.340,179.614,5.774,149.141
C04174=1178.714,-39.723,-43.328,179.612,5.775,149.141
C04175=1178.719,-39.973,-43.317,179.609,5.774,149.142
C04176=1178.724,-40.223,-43.305,179.607,5.774,149.142
C04177=1178.729,-40.472,-43.292,179.604,5.773,149.143
C04178=1178.735,-40.722,-43.280,179.602,5.772,149.144
C04179=1178.740,-40.972,-43.269,179.600,5.773,149.144
C04180=1178.745,-41.222,-43.257,179.597,5.772,149.145
C04181=1178.750,-41.471,-43.244,179.595,5.771,149.145
C04182=1178.756,-41.721,-43.233,179.592,5.771,149.146
C04183=1178.760,-41.971,-43.221,179.590,5.771,149.147
C04184=1178.766,-42.221,-43.209,179.588,5.771,149.147
C04185=1178.771,-42.470,-43.197,179.585,5.770,149.148
C04186=1178.776,-42.720,-43.185,179.583,5.770,149.149
C04187=1178.781,-42.969,-43.174,179.581,5.769,149.149
C04188=1178.787,-43.219,-43.162,179.578,5.768,149.150
C04189=1178.792,-43.469,-43.150,179.576,5.769,149.151
C04190=1178.797,-43.718,-43.138,179.574,5.768,149.151
C04191=1178.802,-43.968,-43.126,179.571,5.768,149.152
C04192=1178.808,-44.218,-43.114,179.568,5.767,149.152
C04193=1178.812,-44.467,-43.103,179.567,5.767,149.153
C04194=1178.818,-44.717,-43.091,179.564,5.767,149.154
C04195=1178.823,-44.967,-43.079,179.561,5.766,149.154
C04196=1178.828,-45.216,-43.067,179.559,5.765,149.155
C04197=1178.833,-45.466,-43.055,179.557,5.765,149.156
C04198=1178.839,-45.715,-43.044,179.555,5.765,149.156
C04199=1178.844,-45.965,-43.033,179.552,5.765,149.157
C04200=1178.849,-46.215,-43.021,179.550,5.764,149.157
C04201=1178.855,-46.465,-43.009,179.547,5.764,149.158
C04202=1178.859,-46.714,-42.998,179.545,5.764,149.159
C04203=1178.865,-46.964,-42.986,179.543,5.763,149.159
C04204=1178.869,-47.214,-42.974,179.540,5.763,149.160
C04205=1178.875,-47.464,-42.962,179.538,5.762,149.160
C04206=1178.881,-47.712,-42.950,179.536,5.762,149.161
C04207=1178.885,-47.962,-42.939,179.533,5.762,149.162
C04208=1178.891,-48.212,-42.927,179.531,5.761,149.162
C04209=1178.895,-48.462,-42.916,179.528,5.761,149.163
C04210=1178.901,-48.712,-42.904,179.526,5.760,149.164
C04211=1178.906,-48.962,-42.892,179.524,5.760,149.164
C04212=1178.911,-49.211,-42.881,179.521,5.760,149.165
C04213=1178.917,-49.481,-42.869,179.519,5.759,149.166
C04214=1178.922,-49.752,-42.856,179.516,5.759,149.166
C04215=1178.928,-50.021,-42.843,179.514,5.758,149.167
C04216=1178.934,-50.292,-42.831,179.511,5.758,149.167
C04217=1178.939,-50.542,-42.819,179.509,5.758,149.168
C04218=1178.944,-50.792,-42.808,179.506,5.758,149.169
C04219=1178.950,-51.041,-42.796,179.504,5.757,149.169
C04220=1178.955,-51.291,-42.785,179.502,5.756,149.170
C04221=1178.960,-51.541,-42.773,179.500,5.757,149.171
C04222=1178.965,-51.790,-42.762,179.497,5.756,149.171
C04223=1178.970,-52.040,-42.750,179.495,5.756,149.172
C04224=1178.975,-52.290,-42.739,179.492,5.755,149.173
C04225=1178.981,-52.539,-42.727,179.490,5.755,149.173
C04226=1178.986,-52.789,-42.716,179.488,5.755,149.174
C04227=1178.991,-53.039,-42.704,179.485,5.754,149.175
C04228=1178.996,-53.289,-42.693,179.483,5.753,149.175
C04229=1179.002,-53.538,-42.682,179.481,5.754,149.176
C04230=1179.007,-53.788,-42.671,179.478,5.753,149.176
C04231=1179.012,-54.038,-42.659,179.476,5.753,149.177
C04232=1179.017,-54.287,-42.647,179.473,5.752,149.178
C04233=1179.022,-54.537,-42.636,179.472,5.752,149.178
C04234=1179.028,-54.786,-42.625,179.469,5.752,149.179
C04235=1179.032,-55.036,-42.613,179.466,5.751,149.179
C04236=1179.038,-55.286,-42.602,179.465,5.751,149.180
C04237=1179.043,-55.536,-42.591,179.462,5.751,149.181
C04238=1179.049,-55.785,-42.579,179.459,5.750,149.181
C04239=1179.054,-56.035,-42.568,179.457,5.750,149.182
C04240=1179.058,-56.285,-42.557,179.455,5.750,149.183
C04241=1179.064,-56.535,-42.546,179.453,5.750,149.183
C04242=1179.069,-56.784,-42.535,179.450,5.749,149.184
C04243=1179.075,-57.034,-42.523,179.448,5.748,149.184
C04244=1179.079,-57.284,-42.512,179.446,5.749,149.185
C04245=1179.084,-57.533,-42.500,179.443,5.748,149.186
C04246=1179.090,-57.783,-42.489,179.441,5.748,149.186
C04247=1179.095,-58.033,-42.478,179.439,5.748,149.187
C04248=1179.101,-58.283,-42.466,179.436,5.747,149.188
C04249=1179.106,-58.532,-42.455,179.434,5.747,149.188
C04250=1179.111,-58.782,-42.445,179.431,5.746,149.189
C04251=1179.116,-59.032,-42.433,179.430,5.746,149.189
C04252=1179.121,-59.281,-42.422,179.427,5.746,149.190
C04253=1179.126,-59.530,-42.411,179.425,5.745,149.191
C04254=1179.132,-59.781,-42.399,179.423,5.745,149.191
C04255=1179.137,-60.030,-42.388,179.420,5.745,149.192
C04256=1179.142,-60.279,-42.377,179.418,5.744,149.192
C04257=1179.148,-60.530,-42.366,179.415,5.744,149.193
C04258=1179.152,-60.780,-42.355,179.413,5.744,149.194
C04259=1179.158,-61.029,-42.344,179.411,5.743,149.194
C04260=1179.163,-61.279,-42.333,179.408,5.743,149.195
C04261=1179.168,-61.529,-42.321,179.406,5.743,149.196
C04262=1179.173,-61.778,-42.310,179.404,5.743,149.196
C04263=1179.178,-62.028,-42.300,179.401,5.742,149.197
C04264=1179.184,-62.278,-42.288,179.399,5.741,149.197
C04265=1179.189,-62.527,-42.277,179.397,5.742,149.198
C04266=1179.194,-62.777,-42.267,179.394,5.741,149.199
C04267=1179.200,-63.027,-42.255,179.392,5.740,149.199
C04268=1179.205,-63.276,-42.244,179.390,5.741,149.200
C04269=1179.210,-63.526,-42.233,179.387,5.740,149.201
C04270=1179.215,-63.776,-42.222,179.385,5.740,149.201
C04271=1179.221,-64.026,-42.211,179.383,5.740,149.202
C04272=1179.226,-64.275,-42.200,179.380,5.740,149.203
C04273=1179.231,-64.525,-42.190,179.378,5.739,149.203
C04274=1179.236,-64.774,-42.178,179.376,5.738,149.204
C04275=1179.241,-65.024,-42.166,179.374,5.738,149.204
C04276=1179.247,-65.274,-42.156,179.371,5.738,149.205
C04277=1179.252,-65.523,-42.145,179.369,5.738,149.206
C04278=1179.257,-65.773,-42.135,179.367,5.738,149.206
C04279=1179.263,-66.023,-42.123,179.364,5.737,149.207
C04280=1179.268,-66.273,-42.112,179.362,5.737,149.208
C04281=1179.273,-66.522,-42.101,179.360,5.737,149.208
C04282=1179.278,-66.772,-42.091,179.357,5.736,149.209
C04283=1179.283,-67.021,-42.080,179.355,5.736,149.209
C04284=1179.289,-67.272,-42.069,179.353,5.736,149.210
C04285=1179.294,-67.521,-42.057,179.351,5.735,149.211
C04286=1179.299,-67.771,-42.047,179.348,5.735,149.211
C04287=1179.304,-68.021,-42.036,179.346,5.735,149.212
C04288=1179.310,-68.270,-42.026,179.344,5.735,149.213
C04289=1179.314,-68.520,-42.014,179.341,5.734,149.213
C04290=1179.321,-68.770,-42.004,179.339,5.734,149.214
C04291=1179.325,-69.019,-41.992,179.337,5.734,149.214
C04292=1179.330,-69.270,-41.982,179.334,5.733,149.215
C04293=1179.336,-69.519,-41.971,179.332,5.733,149.216
C04294=1179.341,-69.769,-41.960,179.330,5.733,149.216
C04295=1179.346,-70.018,-41.950,179.328,5.732,149.217
C04296=1179.351,-70.268,-41.939,179.325,5.732,149.218
C04297=1179.357,-70.518,-41.928,179.323,5.732,149.218
C04298=1179.362,-70.768,-41.917,179.321,5.731,149.219
C04299=1179.367,-71.017,-41.906,179.318,5.731,149.219
C04300=1179.372,-71.267,-41.896,179.316,5.731,149.220
C04301=1179.378,-71.516,-41.885,179.314,5.731,149.221
C04302=1179.383,-71.766,-41.874,179.311,5.730,149.221
C04303=1179.388,-72.016,-41.864,179.309,5.730,149.222
C04304=1179.393,-72.265,-41.853,179.307,5.730,149.223
C04305=1179.399,-72.515,-41.843,179.305,5.729,149.223
C04306=1179.404,-72.766,-41.831,179.302,5.729,149.224
C04307=1179.410,-73.014,-41.820,179.300,5.728,149.224
C04308=1179.415,-73.265,-41.810,179.298,5.729,149.225
C04309=1179.420,-73.514,-41.800,179.296,5.728,149.226
C04310=1179.425,-73.764,-41.788,179.293,5.728,149.226
C04311=1179.431,-74.013,-41.778,179.291,5.728,149.227
C04312=1179.436,-74.264,-41.768,179.289,5.727,149.227
C04313=1179.441,-74.513,-41.757,179.286,5.727,149.228
C04314=1179.446,-74.763,-41.746,179.284,5.727,149.229
C04315=1179.451,-75.012,-41.736,179.282,5.726,149.229
C04316=1179.456,-75.263,-41.725,179.279,5.726,149.230
C04317=1179.463,-75.533,-41.713,179.277,5.726,149.231
C04318=1179.468,-75.804,-41.703,179.275,5.726,149.231
C04319=1179.473,-76.075,-41.690,179.273,5.725,149.232
C04320=1179.480,-76.346,-41.679,179.270,5.725,149.232
C04321=1179.485,-76.596,-41.669,179.267,5.724,149.233
C04322=1179.491,-76.846,-41.658,179.266,5.724,149.234
C04323=1179.495,-77.096,-41.647,179.263,5.724,149.234
C04324=1179.501,-77.345,-41.637,179.261,5.724,149.235
C04325=1179.506,-77.595,-41.626,179.259,5.724,149.236
C04326=1179.511,-77.845,-41.616,179.256,5.723,149.236
C04327=1179.516,-78.095,-41.605,179.254,5.723,149.237
C04328=1179.522,-78.344,-41.595,179.252,5.723,149.237
C04329=1179.527,-78.594,-41.584,179.249,5.722,149.238
C04330=1179.532,-78.844,-41.574,179.247,5.722,149.239
C04331=1179.537,-79.093,-41.564,179.245,5.722,149.239
C04332=1179.542,-79.343,-41.554,179.243,5.721,149.240
C04333=1179.548,-79.593,-41.543,179.240,5.722,149.241
C04334=1179.553,-79.842,-41.533,179.238,5.721,149.241
C04335=1179.558,-80.092,-41.522,179.236,5.721,149.242
C04336=1179.564,-80.342,-41.512,179.234,5.721,149.242
C04337=1179.569,-80.592,-41.501,179.231,5.720,149.243
C04338=1179.574,-80.841,-41.491,179.229,5.720,149.244
C04339=1179.580,-81.091,-41.481,179.227,5.720,149.244
C04340=1179.585,-81.341,-41.470,179.224,5.719,149.245
C04341=1179.590,-81.591,-41.460,179.222,5.720,149.246
C04342=1179.595,-81.841,-41.449,179.220,5.719,149.246
C04343=1179.600,-82.090,-41.440,179.218,5.719,149.247
C04344=1179.606,-82.340,-41.429,179.216,5.718,149.247
C04345=1179.611,-82.589,-41.418,179.213,5.718,149.248
C04346=1179.616,-82.839,-41.408,179.211,5.718,149.249
C04347=1179.621,-83.089,-41.397,179.209,5.718,149.249
C04348=1179.627,-83.339,-41.387,179.206,5.717,149.250
C04349=1179.632,-83.588,-41.377,179.205,5.717,149.250
C04350=1179.637,-83.838,-41.366,179.202,5.717,149.251
C04351=1179.642,-84.088,-41.357,179.200,5.717,149.252
C04352=1179.648,-84.337,-41.347,179.198,5.716,149.252
C04353=1179.653,-84.587,-41.336,179.195,5.716,149.253
C04354=1179.658,-84.837,-41.326,179.193,5.716,149.253
C04355=1179.664,-85.087,-41.316,179.191,5.716,149.254
C04356=1179.669,-85.337,-41.305,179.189,5.715,149.255
C04357=1179.674,-85.586,-41.295,179.187,5.715,149.255
C04358=1179.680,-85.836,-41.285,179.184,5.715,149.256
C04359=1179.685,-86.086,-41.275,179.182,5.715,149.256
C04360=1179.690,-86.335,-41.264,179.180,5.714,149.257
C04361=1179.696,-86.585,-41.254,179.177,5.714,149.258
C04362=1179.700,-86.835,-41.244,179.175,5.714,149.258
C04363=1179.706,-87.084,-41.234,179.173,5.713,149.259
C04364=1179.711,-87.335,-41.225,179.171,5.714,149.260
C04365=1179.716,-87.585,-41.214,179.168,5.713,149.260
C04366=1179.721,-87.834,-41.204,179.166,5.712,149.261
C04367=1179.727,-88.084,-41.194,179.164,5.713,149.261
C04368=1179.732,-88.334,-41.184,179.162,5.712,149.262
C04369=1179.738,-88.583,-41.173,179.160,5.712,149.263
C04370=1179.743,-88.833,-41.163,179.158,5.712,149.263
C04371=1179.748,-89.082,-41.154,179.155,5.711,149.264
C04372=1179.753,-89.332,-41.143,179.153,5.712,149.265
C04373=1179.759,-89.582,-41.133,179.151,5.711,149.265
C04374=1179.764,-89.832,-41.124,179.149,5.711,149.266
C04375=1179.769,-90.082,-41.113,179.146,5.710,149.266
C04376=1179.774,-90.332,-41.103,179.144,5.710,149.267
C04377=1179.780,-90.581,-41.093,179.142,5.710,149.267
C04378=1179.785,-90.830,-41.083,179.139,5.710,149.268
C04379=1179.790,-91.081,-41.073,179.138,5.710,149.269
C04380=1179.796,-91.331,-41.063,179.135,5.709,149.269
C04381=1179.801,-91.580,-41.054,179.133,5.709,149.270
C04382=1179.806,-91.829,-41.043,179.131,5.709,149.271
C04383=1179.811,-92.080,-41.033,179.128,5.708,149.271
C04384=1179.817,-92.329,-41.023,179.127,5.708,149.272
C04385=1179.822,-92.579,-41.014,179.124,5.708,149.272
C04386=1179.828,-92.829,-41.003,179.122,5.708,149.273
C04387=1179.833,-93.079,-40.993,179.120,5.708,149.274
C04388=1179.837,-93.328,-40.983,179.118,5.707,149.274
C04389=1179.843,-93.578,-40.973,179.115,5.707,149.275
C04390=1179.849,-93.828,-40.964,179.113,5.707,149.276
C04391=1179.853,-94.078,-40.954,179.111,5.707,149.276
C04392=1179.859,-94.327,-40.943,179.108,5.707,149.277
C04393=1179.864,-94.577,-40.933,179.106,5.706,149.277
C04394=1179.869,-94.827,-40.924,179.104,5.706,149.278
C04395=1179.875,-95.076,-40.914,179.102,5.705,149.278
C04396=1179.879,-95.326,-40.904,179.100,5.706,149.279
C04397=1179.885,-95.576,-40.895,179.098,5.705,149.280
C04398=1179.891,-95.826,-40.884,179.096,5.705,149.280
C04399=1179.896,-96.075,-40.875,179.093,5.705,149.281
C04400=1179.902,-96.325,-40.865,179.091,5.704,149.282
C04401=1179.907,-96.576,-40.855,179.089,5.705,149.282
C04402=1179.911,-96.825,-40.845,179.087,5.704,149.283
C04403=1179.917,-97.075,-40.836,179.084,5.704,149.283
C04404=1179.922,-97.324,-40.826,179.082,5.703,149.284
C04405=1179.928,-97.574,-40.816,179.080,5.704,149.285
C04406=1179.934,-97.824,-40.806,179.078,5.703,149.285
C04407=1179.938,-98.074,-40.796,179.075,5.703,149.286
C04408=1179.944,-98.323,-40.786,179.074,5.703,149.286
C04409=1179.949,-98.573,-40.777,179.071,5.702,149.287
C04410=1179.954,-98.823,-40.767,179.069,5.702,149.288
C04411=1179.959,-99.072,-40.757,179.067,5.702,149.288
C04412=1179.965,-99.322,-40.748,179.065,5.702,149.289
C04413=1179.970,-99.572,-40.737,179.063,5.702,149.289
C04414=1179.975,-99.822,-40.728,179.061,5.702,149.290
C04415=1179.981,-100.072,-40.718,179.058,5.701,149.291
C04416=1179.986,-100.321,-40.709,179.056,5.700,149.291
C04417=1179.992,-100.571,-40.699,179.054,5.701,149.292
C04418=1179.997,-100.820,-40.689,179.051,5.700,149.293
C04419=1180.002,-101.071,-40.680,179.050,5.700,149.293
C04420=1180.007,-101.321,-40.670,179.047,5.700,149.294
C04421=1180.013,-101.592,-40.660,179.045,5.699,149.294
C04422=1180.019,-101.864,-40.649,179.043,5.700,149.295
C04423=1180.025,-102.136,-40.639,179.040,5.699,149.296
C04424=1180.030,-102.407,-40.628,179.037,5.699,149.296
C04425=1180.036,-102.657,-40.619,179.036,5.699,149.297
C04426=1180.040,-102.907,-40.609,179.033,5.698,149.298
C04427=1180.046,-103.157,-40.600,179.032,5.698,149.298
C04428=1180.051,-103.406,-40.590,179.029,5.698,149.299
C04429=1180.057,-103.656,-40.580,179.027,5.698,149.299
C04430=1180.062,-103.905,-40.571,179.025,5.698,149.300
C04431=1180.067,-104.155,-40.562,179.023,5.698,149.300
C04432=1180.073,-104.405,-40.552,179.020,5.697,149.301
C04433=1180.077,-104.655,-40.542,179.018,5.697,149.302
C04434=1180.083,-104.905,-40.532,179.016,5.697,149.302
C04435=1180.088,-105.155,-40.523,179.014,5.696,149.303
C04436=1180.094,-105.404,-40.513,179.012,5.697,149.304
C04437=1180.099,-105.654,-40.504,179.010,5.696,149.304
C04438=1180.105,-105.904,-40.495,179.007,5.696,149.305
C04439=1180.110,-106.153,-40.485,179.005,5.695,149.305
C04440=1180.115,-106.403,-40.476,179.003,5.696,149.306
C04441=1180.120,-106.653,-40.466,179.001,5.695,149.306
C04442=1180.126,-106.903,-40.457,178.999,5.695,149.307
C04443=1180.131,-107.153,-40.448,178.997,5.695,149.308
C04444=1180.136,-107.402,-40.438,178.995,5.695,149.308
C04445=1180.141,-107.652,-40.429,178.992,5.694,149.309
C04446=1180.147,-107.902,-40.419,178.990,5.694,149.310
C04447=1180.152,-108.151,-40.410,178.988,5.694,149.310
C04448=1180.157,-108.401,-40.401,178.985,5.694,149.311
C04449=1180.163,-108.651,-40.391,178.984,5.694,149.311
C04450=1180.168,-108.901,-40.382,178.981,5.693,149.312
C04451=1180.174,-109.151,-40.373,178.980,5.693,149.312
C04452=1180.178,-109.401,-40.363,178.977,5.693,149.313
C04453=1180.184,-109.651,-40.354,178.975,5.693,149.314
C04454=1180.189,-109.901,-40.344,178.973,5.692,149.314
C04455=1180.194,-110.150,-40.335,178.971,5.692,149.315
C04456=1180.199,-110.400,-40.326,178.969,5.692,149.315
C04457=1180.205,-110.650,-40.316,178.967,5.692,149.316
C04458=1180.210,-110.899,-40.307,178.965,5.691,149.317
C04459=1180.215,-111.149,-40.298,178.963,5.692,149.317
C04460=1180.221,-111.399,-40.288,178.960,5.691,149.318
C04461=1180.226,-111.648,-40.279,178.958,5.691,149.318
C04462=1180.231,-111.898,-40.270,178.956,5.691,149.319
C04463=1180.237,-112.148,-40.260,178.953,5.690,149.320
C04464=1180.242,-112.398,-40.251,178.952,5.690,149.320
C04465=1180.248,-112.647,-40.242,178.949,5.690,149.321
C04466=1180.253,-112.897,-40.233,178.947,5.690,149.321
C04467=1180.259,-113.147,-40.224,178.945,5.690,149.322
C04468=1180.264,-113.397,-40.215,178.943,5.690,149.323
C04469=1180.269,-113.646,-40.205,178.941,5.689,149.323
C04470=1180.275,-113.896,-40.196,178.939,5.689,149.324
C04471=1180.280,-114.146,-40.187,178.936,5.689,149.324
C04472=1180.285,-114.396,-40.178,178.935,5.689,149.325
C04473=1180.290,-114.646,-40.169,178.932,5.688,149.326
C04474=1180.296,-114.895,-40.159,178.930,5.688,149.326
C04475=1180.301,-115.145,-40.150,178.928,5.688,149.327
C04476=1180.306,-115.395,-40.141,178.926,5.688,149.327
C04477=1180.311,-115.645,-40.132,178.924,5.687,149.328
C04478=1180.317,-115.895,-40.123,178.922,5.688,149.329
C04479=1180.322,-116.145,-40.114,178.920,5.687,149.329
C04480=1180.327,-116.394,-40.104,178.918,5.687,149.330
C04481=1180.333,-116.644,-40.095,178.915,5.687,149.330
C04482=1180.338,-116.894,-40.086,178.913,5.687,149.331
C04483=1180.344,-117.144,-40.077,178.911,5.686,149.331
C04484=1180.349,-117.393,-40.068,178.909,5.687,149.332
C04485=1180.355,-117.643,-40.059,178.907,5.686,149.333
C04486=1180.360,-117.893,-40.050,178.905,5.686,149.333
C04487=1180.365,-118.142,-40.040,178.903,5.686,149.334
C04488=1180.370,-118.392,-40.031,178.901,5.686,149.334
C04489=1180.376,-118.642,-40.022,178.898,5.685,149.335
C04490=1180.381,-118.892,-40.014,178.897,5.685,149.335
C04491=1180.386,-119.142,-40.005,178.894,5.685,149.336
C04492=1180.392,-119.392,-39.995,178.892,5.685,149.337
C04493=1180.397,-119.642,-39.986,178.890,5.684,149.337
C04494=1180.403,-119.891,-39.978,178.888,5.684,149.338
C04495=1180.408,-120.141,-39.969,178.886,5.684,149.338
C04496=1180.413,-120.391,-39.960,178.884,5.684,149.339
C04497=1180.418,-120.640,-39.951,178.882,5.683,149.340
C04498=1180.423,-120.890,-39.942,178.880,5.684,149.340
C04499=1180.429,-121.140,-39.933,178.877,5.683,149.341
C04500=1180.435,-121.390,-39.924,178.875,5.683,149.342
C04501=1180.440,-121.640,-39.915,178.873,5.683,149.342
C04502=1180.445,-121.889,-39.906,178.871,5.683,149.342
C04503=1180.451,-122.139,-39.897,178.869,5.682,149.343
C04504=1180.456,-122.389,-39.888,178.867,5.682,149.344
C04505=1180.461,-122.639,-39.880,178.865,5.682,149.344
C04506=1180.466,-122.889,-39.871,178.863,5.682,149.345
C04507=1180.471,-123.139,-39.862,178.860,5.682,149.346
C04508=1180.477,-123.389,-39.852,178.859,5.682,149.346
C04509=1180.483,-123.638,-39.844,178.856,5.681,149.347
C04510=1180.488,-123.888,-39.835,178.854,5.681,149.347
C04511=1180.493,-124.138,-39.826,178.852,5.680,149.348
C04512=1180.498,-124.387,-39.817,178.850,5.681,149.348
C04513=1180.504,-124.637,-39.808,178.848,5.680,149.349
C04514=1180.509,-124.887,-39.799,178.846,5.680,149.349
C04515=1180.515,-125.136,-39.791,178.844,5.680,149.350
C04516=1180.520,-125.386,-39.782,178.842,5.680,149.351
C04517=1180.525,-125.636,-39.773,178.840,5.680,149.351
C04518=1180.530,-125.886,-39.764,178.838,5.679,149.352
C04519=1180.535,-126.136,-39.755,178.836,5.680,149.353
C04520=1180.541,-126.385,-39.747,178.833,5.679,149.353
C04521=1180.546,-126.635,-39.738,178.832,5.679,149.354
C04522=1180.552,-126.885,-39.730,178.829,5.679,149.354
C04523=1180.557,-127.135,-39.721,178.828,5.679,149.355
C04524=1180.563,-127.385,-39.711,178.825,5.678,149.355
C04525=1180.142,-127.396,-39.752,178.821,5.682,149.357
C04526=1180.136,-127.146,-39.760,178.824,5.682,149.357
C04527=1180.131,-126.897,-39.769,178.825,5.682,149.356
C04528=1180.125,-126.646,-39.777,178.828,5.682,149.355
C04529=1180.120,-126.396,-39.786,178.830,5.682,149.355
C04530=1180.115,-126.147,-39.795,178.832,5.683,149.354
C04531=1180.109,-125.896,-39.804,178.834,5.683,149.354
C04532=1180.103,-125.647,-39.813,178.836,5.683,149.353
C04533=1180.098,-125.397,-39.822,178.838,5.683,149.353
C04534=1180.093,-125.148,-39.831,178.840,5.684,149.352
C04535=1180.088,-124.898,-39.840,178.842,5.684,149.352
C04536=1180.083,-124.648,-39.849,178.845,5.684,149.351
C04537=1180.077,-124.398,-39.857,178.846,5.684,149.350
C04538=1180.072,-124.149,-39.866,178.849,5.684,149.350
C04539=1180.066,-123.899,-39.875,178.850,5.684,149.349
C04540=1180.061,-123.649,-39.884,178.853,5.685,149.348
C04541=1180.056,-123.399,-39.892,178.855,5.685,149.348
C04542=1180.051,-123.149,-39.901,178.857,5.686,149.347
C04543=1180.045,-122.899,-39.910,178.859,5.685,149.347
C04544=1180.040,-122.650,-39.918,178.861,5.686,149.346
C04545=1180.034,-122.400,-39.928,178.863,5.686,149.346
C04546=1180.029,-122.150,-39.937,178.865,5.685,149.345
C04547=1180.023,-121.900,-39.946,178.867,5.686,149.345
C04548=1180.018,-121.650,-39.955,178.869,5.686,149.344
C04549=1180.013,-121.400,-39.963,178.871,5.687,149.343
C04550=1180.008,-121.150,-39.972,178.873,5.686,149.343
C04551=1180.002,-120.902,-39.982,178.876,5.687,149.342
C04552=1179.997,-120.652,-39.990,178.878,5.687,149.341
C04553=1179.991,-120.402,-40.000,178.880,5.687,149.341
C04554=1179.986,-120.152,-40.009,178.882,5.687,149.340
C04555=1179.981,-119.902,-40.018,178.884,5.688,149.340
C04556=1179.976,-119.652,-40.027,178.886,5.688,149.339
C04557=1179.971,-119.402,-40.036,178.888,5.688,149.339
C04558=1179.966,-119.153,-40.044,178.890,5.688,149.338
C04559=1179.960,-118.902,-40.054,178.893,5.688,149.337
C04560=1179.954,-118.653,-40.062,178.894,5.688,149.337
C04561=1179.949,-118.403,-40.071,178.897,5.689,149.336
C04562=1179.944,-118.154,-40.080,178.899,5.689,149.336
C04563=1179.938,-117.904,-40.089,178.901,5.689,149.335
C04564=1179.934,-117.654,-40.099,178.903,5.689,149.334
C04565=1179.928,-117.404,-40.108,178.905,5.690,149.334
C04566=1179.922,-117.154,-40.117,178.907,5.689,149.333
C04567=1179.917,-116.905,-40.126,178.909,5.690,149.333
C04568=1179.912,-116.655,-40.135,178.911,5.690,149.332
C04569=1179.907,-116.405,-40.144,178.914,5.691,149.332
C04570=1179.901,-116.155,-40.153,178.915,5.691,149.331
C04571=1179.896,-115.905,-40.162,178.918,5.691,149.330
C04572=1179.890,-115.656,-40.171,178.920,5.691,149.330
C04573=1179.885,-115.407,-40.180,178.922,5.691,149.329
C04574=1179.879,-115.156,-40.190,178.924,5.692,149.329
C04575=1179.874,-114.906,-40.199,178.926,5.692,149.328
C04576=1179.869,-114.657,-40.208,178.929,5.692,149.327
C04577=1179.864,-114.407,-40.217,178.931,5.692,149.327
C04578=1179.858,-114.157,-40.227,178.933,5.693,149.326
C04579=1179.853,-113.907,-40.236,178.935,5.692,149.326
C04580=1179.848,-113.658,-40.245,178.937,5.693,149.325
C04581=1179.842,-113.407,-40.254,178.939,5.693,149.324
C04582=1179.837,-113.158,-40.264,178.942,5.694,149.324
C04583=1179.832,-112.908,-40.273,178.943,5.694,149.323
C04584=1179.827,-112.658,-40.281,178.946,5.694,149.323
C04585=1179.821,-112.408,-40.291,178.947,5.694,149.322
C04586=1179.816,-112.159,-40.301,178.950,5.694,149.321
C04587=1179.811,-111.909,-40.309,178.952,5.694,149.321
C04588=1179.805,-111.659,-40.319,178.954,5.695,149.320
C04589=1179.800,-111.409,-40.328,178.956,5.695,149.320
C04590=1179.795,-111.160,-40.337,178.959,5.695,149.319
C04591=1179.789,-110.910,-40.347,178.960,5.695,149.319
C04592=1179.784,-110.660,-40.356,178.963,5.695,149.318
C04593=1179.779,-110.411,-40.366,178.964,5.695,149.317
C04594=1179.773,-110.161,-40.375,178.967,5.696,149.317
C04595=1179.768,-109.911,-40.384,178.969,5.696,149.316
C04596=1179.763,-109.661,-40.394,178.971,5.696,149.315
C04597=1179.757,-109.411,-40.403,178.973,5.696,149.315
C04598=1179.752,-109.161,-40.412,178.976,5.696,149.314
C04599=1179.747,-108.912,-40.422,178.978,5.697,149.314
C04600=1179.741,-108.662,-40.431,178.980,5.697,149.313
C04601=1179.736,-108.412,-40.440,178.982,5.698,149.313
C04602=1179.731,-108.163,-40.450,178.984,5.697,149.312
C04603=1179.725,-107.913,-40.459,178.986,5.698,149.311
C04604=1179.720,-107.663,-40.468,178.988,5.698,149.311
C04605=1179.715,-107.413,-40.478,178.991,5.698,149.310
C04606=1179.709,-107.164,-40.487,178.992,5.698,149.310
C04607=1179.704,-106.914,-40.496,178.995,5.699,149.309
C04608=1179.699,-106.664,-40.506,178.997,5.699,149.309
C04609=1179.693,-106.414,-40.515,178.999,5.699,149.308
C04610=1179.688,-106.165,-40.525,179.001,5.699,149.307
C04611=1179.683,-105.915,-40.534,179.004,5.699,149.307
C04612=1179.678,-105.666,-40.544,179.006,5.700,149.306
C04613=1179.673,-105.415,-40.554,179.008,5.700,149.305
C04614=1179.667,-105.165,-40.562,179.010,5.701,149.305
C04615=1179.662,-104.915,-40.573,179.012,5.700,149.304
C04616=1179.657,-104.666,-40.582,179.014,5.701,149.304
C04617=1179.651,-104.416,-40.592,179.016,5.701,149.303
C04618=1179.646,-104.166,-40.601,179.019,5.701,149.303
C04619=1179.641,-103.917,-40.610,179.021,5.701,149.302
C04620=1179.635,-103.667,-40.620,179.023,5.702,149.301
C04621=1179.630,-103.418,-40.629,179.025,5.701,149.301
C04622=1179.624,-103.167,-40.639,179.027,5.702,149.300
C04623=1179.619,-102.918,-40.649,179.030,5.702,149.299
C04624=1179.614,-102.667,-40.658,179.031,5.702,149.299
C04625=1179.609,-102.418,-40.668,179.034,5.703,149.298
C04626=1179.603,-102.147,-40.678,179.036,5.702,149.297
C04627=1179.597,-101.875,-40.689,179.038,5.703,149.297
C04628=1179.591,-101.603,-40.699,179.041,5.704,149.296
C04629=1179.586,-101.331,-40.710,179.043,5.703,149.296
C04630=1179.580,-101.081,-40.719,179.045,5.704,149.295
C04631=1179.576,-100.832,-40.729,179.048,5.704,149.294
C04632=1179.570,-100.582,-40.738,179.050,5.704,149.294
C04633=1179.565,-100.333,-40.748,179.052,5.705,149.293
C04634=1179.559,-100.082,-40.758,179.054,5.704,149.292
C04635=1179.555,-99.833,-40.768,179.057,5.705,149.292
C04636=1179.549,-99.583,-40.778,179.059,5.705,149.291
C04637=1179.544,-99.333,-40.787,179.061,5.705,149.291
C04638=1179.538,-99.084,-40.797,179.063,5.705,149.290
C04639=1179.532,-98.833,-40.806,179.065,5.706,149.290
C04640=1179.527,-98.584,-40.816,179.068,5.706,149.289
C04641=1179.522,-98.335,-40.826,179.069,5.706,149.288
C04642=1179.517,-98.084,-40.835,179.072,5.707,149.288
C04643=1179.512,-97.835,-40.846,179.074,5.707,149.287
C04644=1179.507,-97.585,-40.855,179.076,5.707,149.286
C04645=1179.501,-97.335,-40.865,179.078,5.707,149.286
C04646=1179.495,-97.086,-40.875,179.081,5.707,149.285
C04647=1179.490,-96.836,-40.884,179.083,5.708,149.285
C04648=1179.485,-96.585,-40.894,179.085,5.708,149.284
C04649=1179.480,-96.336,-40.904,179.087,5.709,149.284
C04650=1179.475,-96.087,-40.914,179.089,5.708,149.283
C04651=1179.469,-95.837,-40.924,179.092,5.709,149.282
C04652=1179.464,-95.587,-40.933,179.093,5.709,149.282
C04653=1179.459,-95.337,-40.944,179.096,5.709,149.281
C04654=1179.454,-95.087,-40.953,179.098,5.710,149.281
C04655=1179.448,-94.838,-40.963,179.100,5.709,149.280
C04656=1179.443,-94.588,-40.973,179.103,5.710,149.279
C04657=1179.437,-94.338,-40.982,179.105,5.710,149.279
C04658=1179.432,-94.088,-40.993,179.107,5.710,149.278
C04659=1179.427,-93.839,-41.003,179.109,5.710,149.277
C04660=1179.422,-93.589,-41.013,179.111,5.711,149.277
C04661=1179.416,-93.339,-41.022,179.114,5.711,149.276
C04662=1179.410,-93.090,-41.032,179.115,5.711,149.276
C04663=1179.406,-92.840,-41.042,179.118,5.712,149.275
C04664=1179.401,-92.590,-41.052,179.120,5.711,149.274
C04665=1179.395,-92.341,-41.063,179.122,5.712,149.274
C04666=1179.390,-92.091,-41.072,179.125,5.712,149.273
C04667=1179.385,-91.840,-41.082,179.127,5.712,149.273
C04668=1179.379,-91.591,-41.092,179.129,5.713,149.272
C04669=1179.374,-91.342,-41.102,179.131,5.713,149.271
C04670=1179.369,-91.092,-41.112,179.133,5.713,149.271
C04671=1179.364,-90.841,-41.122,179.136,5.714,149.270
C04672=1179.358,-90.592,-41.132,179.138,5.714,149.270
C04673=1179.353,-90.343,-41.142,179.140,5.714,149.269
C04674=1179.347,-90.093,-41.152,179.142,5.714,149.268
C04675=1179.342,-89.843,-41.163,179.145,5.714,149.268
C04676=1179.337,-89.593,-41.173,179.147,5.715,149.267
C04677=1179.332,-89.343,-41.182,179.149,5.715,149.266
C04678=1179.327,-89.093,-41.192,179.151,5.716,149.266
C04679=1179.321,-88.844,-41.202,179.153,5.715,149.265
C04680=1179.316,-88.594,-41.212,179.155,5.716,149.265
C04681=1179.311,-88.345,-41.222,179.158,5.716,149.264
C04682=1179.306,-88.095,-41.233,179.160,5.716,149.263
C04683=1179.300,-87.845,-41.243,179.162,5.717,149.263
C04684=1179.294,-87.595,-41.253,179.164,5.716,149.262
C04685=1179.290,-87.345,-41.263,179.167,5.717,149.262
C04686=1179.285,-87.096,-41.274,179.169,5.718,149.261
C04687=1179.279,-86.846,-41.283,179.171,5.718,149.260
C04688=1179.274,-86.596,-41.294,179.174,5.718,149.260
C04689=1179.269,-86.346,-41.303,179.176,5.718,149.259
C04690=1179.263,-86.097,-41.313,179.178,5.718,149.259
C04691=1179.258,-85.847,-41.324,179.181,5.719,149.258
C04692=1179.253,-85.597,-41.334,179.182,5.719,149.257
C04693=1179.247,-85.347,-41.344,179.185,5.719,149.257
C04694=1179.243,-85.097,-41.354,179.186,5.719,149.256
C04695=1179.237,-84.848,-41.365,179.189,5.720,149.255
C04696=1179.232,-84.598,-41.375,179.192,5.720,149.255
C04697=1179.227,-84.348,-41.385,179.193,5.720,149.254
C04698=1179.221,-84.099,-41.396,179.196,5.720,149.254
C04699=1179.215,-83.849,-41.406,179.198,5.720,149.253
C04700=1179.211,-83.599,-41.416,179.200,5.721,149.252
C04701=1179.206,-83.350,-41.426,179.202,5.722,149.252
C04702=1179.200,-83.100,-41.436,179.205,5.721,149.251
C04703=1179.195,-82.850,-41.447,179.207,5.722,149.250
C04704=1179.189,-82.600,-41.457,179.209,5.722,149.250
C04705=1179.184,-82.350,-41.468,179.211,5.722,149.249
C04706=1179.179,-82.101,-41.478,179.214,5.723,149.249
C04707=1179.173,-81.852,-41.489,179.216,5.722,149.248
C04708=1179.169,-81.602,-41.499,179.218,5.723,149.247
C04709=1179.164,-81.352,-41.509,179.221,5.724,149.247
C04710=1179.158,-81.103,-41.519,179.223,5.723,149.246
C04711=1179.153,-80.852,-41.530,179.225,5.724,149.246
C04712=1179.147,-80.603,-41.540,179.228,5.724,149.245
C04713=1179.142,-80.353,-41.550,179.229,5.724,149.245
C04714=1179.137,-80.103,-41.561,179.232,5.725,149.244
C04715=1179.131,-79.853,-41.571,179.234,5.724,149.243
C04716=1179.126,-79.604,-41.582,179.236,5.725,149.243
C04717=1179.121,-79.354,-41.592,179.239,5.726,149.242
C04718=1179.116,-79.104,-41.603,179.240,5.726,149.241
C04719=1179.110,-78.854,-41.613,179.243,5.726,149.241
C04720=1179.105,-78.604,-41.624,179.246,5.726,149.240
C04721=1179.100,-78.355,-41.633,179.247,5.726,149.240
C04722=1179.095,-78.106,-41.644,179.250,5.727,149.239
C04723=1179.090,-77.856,-41.655,179.252,5.728,149.238
C04724=1179.085,-77.606,-41.665,179.254,5.727,149.238
C04725=1179.080,-77.356,-41.676,179.257,5.728,149.237
C04726=1179.074,-77.106,-41.686,179.259,5.728,149.236
C04727=1179.069,-76.856,-41.696,179.261,5.728,149.236
C04728=1179.064,-76.607,-41.707,179.263,5.729,149.235
C04729=1179.058,-76.358,-41.717,179.265,5.728,149.235
C04730=1179.052,-76.086,-41.729,179.268,5.729,149.234
C04731=1179.047,-75.815,-41.741,179.271,5.729,149.233
C04732=1179.041,-75.545,-41.752,179.273,5.730,149.233
C04733=1179.035,-75.273,-41.763,179.276,5.730,149.232
C04734=1179.030,-75.023,-41.775,179.278,5.730,149.231
C04735=1179.025,-74.774,-41.785,179.280,5.731,149.231
C04736=1179.020,-74.524,-41.795,179.283,5.731,149.230
C04737=1179.014,-74.275,-41.806,179.285,5.731,149.229
C04738=1179.009,-74.025,-41.817,179.287,5.732,149.229
C04739=1179.004,-73.775,-41.827,179.290,5.732,149.228
C04740=1178.998,-73.525,-41.837,179.291,5.732,149.228
C04741=1178.993,-73.276,-41.849,179.294,5.732,149.227
C04742=1178.988,-73.026,-41.859,179.296,5.733,149.226
C04743=1178.983,-72.776,-41.869,179.298,5.733,149.226
C04744=1178.977,-72.527,-41.881,179.301,5.733,149.225
C04745=1178.972,-72.276,-41.892,179.303,5.734,149.224
C04746=1178.966,-72.027,-41.902,179.305,5.734,149.224
C04747=1178.961,-71.777,-41.913,179.308,5.734,149.223
C04748=1178.956,-71.528,-41.923,179.309,5.734,149.223
C04749=1178.951,-71.277,-41.934,179.312,5.734,149.222
C04750=1178.946,-71.028,-41.945,179.315,5.735,149.221
C04751=1178.941,-70.778,-41.955,179.317,5.736,149.221
C04752=1178.936,-70.529,-41.967,179.319,5.735,149.220
C04753=1178.930,-70.279,-41.977,179.321,5.736,149.220
C04754=1178.925,-70.029,-41.988,179.324,5.736,149.219
C04755=1178.919,-69.780,-41.999,179.326,5.736,149.218
C04756=1178.914,-69.529,-42.009,179.328,5.737,149.218
C04757=1178.909,-69.280,-42.020,179.331,5.737,149.217
C04758=1178.904,-69.030,-42.031,179.333,5.737,149.216
C04759=1178.899,-68.781,-42.042,179.335,5.738,149.216
C04760=1178.894,-68.531,-42.052,179.338,5.738,149.215
C04761=1178.887,-68.281,-42.063,179.339,5.738,149.215
C04762=1178.883,-68.032,-42.075,179.342,5.739,149.214
C04763=1178.878,-67.781,-42.085,179.345,5.739,149.213
C04764=1178.872,-67.532,-42.096,179.346,5.739,149.213
C04765=1178.867,-67.282,-42.107,179.349,5.739,149.212
C04766=1178.861,-67.033,-42.118,179.351,5.740,149.212
C04767=1178.856,-66.783,-42.129,179.353,5.740,149.211
C04768=1178.852,-66.533,-42.140,179.356,5.740,149.210
C04769=1178.846,-66.284,-42.150,179.358,5.741,149.210
C04770=1178.841,-66.034,-42.162,179.360,5.741,149.209
C04771=1178.835,-65.784,-42.172,179.363,5.741,149.208
C04772=1178.830,-65.534,-42.184,179.365,5.742,149.208
C04773=1178.825,-65.284,-42.194,179.367,5.741,149.207
C04774=1178.820,-65.035,-42.205,179.370,5.742,149.206
C04775=1178.815,-64.786,-42.216,179.372,5.743,149.206
C04776=1178.809,-64.536,-42.227,179.374,5.743,149.205
C04777=1178.804,-64.286,-42.239,179.376,5.743,149.205
C04778=1178.799,-64.036,-42.249,179.379,5.744,149.204
C04779=1178.794,-63.787,-42.260,179.381,5.744,149.203
C04780=1178.788,-63.536,-42.271,179.383,5.744,149.203
C04781=1178.784,-63.287,-42.282,179.386,5.744,149.202
C04782=1178.778,-63.038,-42.293,179.388,5.745,149.201
C04783=1178.773,-62.787,-42.305,179.390,5.745,149.201
C04784=1178.767,-62.538,-42.315,179.393,5.745,149.200
C04785=1178.762,-62.288,-42.326,179.395,5.746,149.200
C04786=1178.758,-62.039,-42.337,179.397,5.746,149.199
C04787=1178.752,-61.789,-42.349,179.400,5.746,149.198
C04788=1178.747,-61.539,-42.359,179.402,5.747,149.198
C04789=1178.742,-61.289,-42.371,179.404,5.747,149.197
C04790=1178.736,-61.040,-42.382,179.406,5.747,149.196
C04791=1178.731,-60.790,-42.393,179.409,5.748,149.196
C04792=1178.726,-60.540,-42.404,179.411,5.748,149.195
C04793=1178.720,-60.291,-42.416,179.413,5.748,149.195
C04794=1178.715,-60.041,-42.426,179.416,5.749,149.194
C04795=1178.710,-59.791,-42.438,179.418,5.749,149.193
C04796=1178.705,-59.541,-42.449,179.420,5.750,149.193
C04797=1178.700,-59.292,-42.460,179.422,5.749,149.192
C04798=1178.695,-59.042,-42.471,179.425,5.750,149.191
C04799=1178.689,-58.792,-42.483,179.427,5.751,149.191
C04800=1178.684,-58.543,-42.494,179.430,5.751,149.190
C04801=1178.679,-58.293,-42.504,179.432,5.751,149.190
C04802=1178.674,-58.043,-42.516,179.434,5.751,149.189
C04803=1178.668,-57.794,-42.527,179.437,5.752,149.188
C04804=1178.664,-57.545,-42.538,179.439,5.751,149.188
C04805=1178.658,-57.295,-42.550,179.441,5.752,149.187
C04806=1178.653,-57.044,-42.561,179.444,5.753,149.187
C04807=1178.647,-56.795,-42.572,179.447,5.753,149.186
C04808=1178.642,-56.545,-42.584,179.448,5.753,149.185
C04809=1178.638,-56.296,-42.595,179.451,5.754,149.185
C04810=1178.632,-56.046,-42.607,179.453,5.754,149.184
C04811=1178.627,-55.796,-42.617,179.455,5.754,149.183
C04812=1178.621,-55.546,-42.629,179.458,5.754,149.183
C04813=1178.617,-55.297,-42.640,179.460,5.755,149.182
C04814=1178.612,-55.047,-42.651,179.463,5.756,149.182
C04815=1178.606,-54.798,-42.663,179.465,5.755,149.181
C04816=1178.601,-54.548,-42.674,179.467,5.756,149.180
C04817=1178.595,-54.298,-42.685,179.470,5.757,149.180
C04818=1178.591,-54.048,-42.697,179.472,5.757,149.179
C04819=1178.585,-53.799,-42.708,179.474,5.757,149.179
C04820=1178.580,-53.549,-42.720,179.476,5.757,149.178
C04821=1178.575,-53.299,-42.731,179.479,5.758,149.177
C04822=1178.570,-53.050,-42.743,179.481,5.759,149.177
C04823=1178.564,-52.800,-42.755,179.483,5.758,149.176
C04824=1178.559,-52.551,-42.766,179.486,5.759,149.175
C04825=1178.554,-52.301,-42.777,179.488,5.759,149.175
C04826=1178.549,-52.051,-42.788,179.491,5.760,149.174
C04827=1178.543,-51.801,-42.800,179.492,5.760,149.174
C04828=1178.539,-51.551,-42.811,179.495,5.760,149.173
C04829=1178.533,-51.302,-42.823,179.498,5.761,149.172
C04830=1178.528,-51.052,-42.834,179.500,5.762,149.172
C04831=1178.522,-50.802,-42.846,179.502,5.761,149.171
C04832=1178.518,-50.553,-42.857,179.505,5.762,149.170
C04833=1178.512,-50.303,-42.869,179.507,5.762,149.170
C04834=1178.506,-50.033,-42.882,179.510,5.763,149.169
C04835=1178.501,-49.762,-42.894,179.512,5.763,149.168
C04836=1178.495,-49.492,-42.907,179.515,5.764,149.168
C04837=1178.489,-49.221,-42.919,179.517,5.763,149.167
C04838=1178.485,-48.972,-42.930,179.520,5.764,149.166
C04839=1178.479,-48.723,-42.943,179.522,5.765,149.166
C04840=1178.475,-48.473,-42.954,179.525,5.765,149.165
C04841=1178.469,-48.224,-42.965,179.527,5.765,149.164
C04842=1178.464,-47.974,-42.977,179.529,5.765,149.164
C04843=1178.459,-47.724,-42.989,179.531,5.766,149.163
C04844=1178.453,-47.474,-43.001,179.534,5.766,149.163
C04845=1178.449,-47.225,-43.012,179.536,5.767,149.162
C04846=1178.443,-46.975,-43.024,179.538,5.767,149.161
C04847=1178.438,-46.725,-43.035,179.541,5.768,149.161
C04848=1178.432,-46.476,-43.047,179.543,5.768,149.160
C04849=1178.427,-46.226,-43.058,179.546,5.768,149.159
C04850=1178.422,-45.976,-43.070,179.547,5.768,149.159
C04851=1178.417,-45.726,-43.082,179.550,5.769,149.158
C04852=1178.411,-45.476,-43.093,179.553,5.769,149.158
C04853=1178.407,-45.227,-43.105,179.555,5.770,149.157
C04854=1178.402,-44.977,-43.117,179.558,5.771,149.156
C04855=1178.396,-44.727,-43.129,179.560,5.770,149.156
C04856=1178.391,-44.478,-43.141,179.562,5.771,149.155
C04857=1178.386,-44.228,-43.152,179.565,5.771,149.155
C04858=1178.380,-43.979,-43.164,179.567,5.772,149.154
C04859=1178.376,-43.730,-43.176,179.569,5.772,149.153
C04860=1178.370,-43.480,-43.188,179.571,5.772,149.153
C04861=1178.365,-43.230,-43.200,179.574,5.773,149.152
C04862=1178.360,-42.980,-43.211,179.576,5.774,149.151
C04863=1178.355,-42.730,-43.223,179.579,5.774,149.151
C04864=1178.349,-42.481,-43.235,179.581,5.774,149.150
C04865=1178.345,-42.231,-43.247,179.583,5.774,149.150
C04866=1178.339,-41.981,-43.259,179.586,5.775,149.149
C04867=1178.334,-41.731,-43.271,179.589,5.775,149.148
C04868=1178.329,-41.481,-43.282,179.591,5.776,149.148
C04869=1178.324,-41.232,-43.294,179.593,5.776,149.147
C04870=1178.319,-40.983,-43.306,179.595,5.776,149.146
C04871=1178.313,-40.733,-43.318,179.598,5.777,149.146
C04872=1178.308,-40.483,-43.331,179.600,5.777,149.145
C04873=1178.303,-40.234,-43.342,179.603,5.778,149.144
C04874=1178.297,-39.984,-43.354,179.605,5.778,149.144
C04875=1178.292,-39.734,-43.365,179.607,5.778,149.143
C04876=1178.287,-39.485,-43.378,179.610,5.779,149.143
C04877=1178.282,-39.236,-43.389,179.612,5.780,149.142
C04878=1178.277,-38.986,-43.401,179.615,5.780,149.141
C04879=1178.272,-38.736,-43.414,179.617,5.780,149.141
C04880=1178.266,-38.486,-43.426,179.619,5.780,149.140
C04881=1178.261,-38.236,-43.438,179.622,5.781,149.140
C04882=1178.256,-37.987,-43.450,179.624,5.781,149.139
C04883=1178.251,-37.737,-43.462,179.627,5.782,149.138
C04884=1178.246,-37.488,-43.473,179.629,5.782,149.138
C04885=1178.240,-37.238,-43.486,179.631,5.782,149.137
C04886=1178.235,-36.988,-43.498,179.633,5.783,149.136
C04887=1178.230,-36.738,-43.510,179.636,5.783,149.136
C04888=1178.225,-36.489,-43.522,179.639,5.784,149.135
C04889=1178.220,-36.239,-43.534,179.640,5.784,149.135
C04890=1178.215,-35.990,-43.546,179.643,5.784,149.134
C04891=1178.209,-35.740,-43.558,179.646,5.785,149.133
C04892=1178.204,-35.491,-43.571,179.648,5.786,149.133
C04893=1178.199,-35.241,-43.583,179.651,5.786,149.132
C04894=1178.193,-34.991,-43.595,179.653,5.786,149.131
C04895=1178.189,-34.741,-43.607,179.655,5.786,149.131
C04896=1178.184,-34.491,-43.619,179.657,5.787,149.130
C04897=1178.179,-34.242,-43.631,179.660,5.787,149.129
C04898=1178.173,-33.992,-43.643,179.663,5.788,149.129
C04899=1178.168,-33.743,-43.656,179.665,5.789,149.128
C04900=1178.163,-33.493,-43.668,179.668,5.789,149.128
C04901=1178.158,-33.243,-43.680,179.670,5.789,149.127
C04902=1178.152,-32.994,-43.692,179.672,5.790,149.126
C04903=1178.147,-32.744,-43.705,179.675,5.790,149.126
C04904=1178.142,-32.494,-43.717,179.677,5.790,149.125
C04905=1178.137,-32.245,-43.729,179.679,5.791,149.125
C04906=1178.132,-31.995,-43.741,179.682,5.792,149.124
C04907=1178.127,-31.746,-43.753,179.684,5.791,149.123
C04908=1178.121,-31.496,-43.765,179.686,5.792,149.123
C04909=1178.116,-31.247,-43.778,179.689,5.793,149.122
C04910=1178.111,-30.996,-43.790,179.692,5.793,149.121
C04911=1178.106,-30.747,-43.803,179.694,5.794,149.121
C04912=1178.101,-30.497,-43.815,179.696,5.794,149.120
C04913=1178.096,-30.248,-43.827,179.699,5.794,149.119
C04914=1178.091,-29.998,-43.840,179.701,5.795,149.119
C04915=1178.085,-29.748,-43.852,179.703,5.795,149.118
C04916=1178.080,-29.499,-43.864,179.706,5.796,149.118
C04917=1178.075,-29.250,-43.877,179.708,5.796,149.117
C04918=1178.070,-28.999,-43.889,179.711,5.797,149.116
C04919=1178.065,-28.750,-43.902,179.714,5.797,149.116
C04920=1178.060,-28.500,-43.914,179.715,5.797,149.115
C04921=1178.054,-28.250,-43.926,179.718,5.798,149.115
C04922=1178.049,-28.001,-43.939,179.720,5.798,149.114
C04923=1178.044,-27.751,-43.951,179.723,5.799,149.113
C04924=1178.039,-27.502,-43.963,179.725,5.800,149.113
C04925=1178.034,-27.252,-43.976,179.728,5.800,149.112
C04926=1178.029,-27.003,-43.989,179.730,5.801,149.112
C04927=1178.024,-26.753,-44.001,179.732,5.800,149.111
C04928=1178.019,-26.503,-44.013,179.735,5.801,149.110
C04929=1178.013,-26.254,-44.026,179.737,5.802,149.110
C04930=1178.008,-26.004,-44.038,179.740,5.802,149.109
C04931=1178.003,-25.754,-44.051,179.742,5.803,149.108
C04932=1177.998,-25.504,-44.064,179.745,5.803,149.108
C04933=1177.993,-25.255,-44.076,179.747,5.804,149.107
C04934=1177.987,-25.005,-44.088,179.749,5.803,149.106
C04935=1177.982,-24.756,-44.101,179.751,5.804,149.106
C04936=1177.977,-24.506,-44.114,179.754,5.805,149.105
C04937=1177.972,-24.256,-44.127,179.757,5.805,149.105
C04938=1177.966,-23.987,-44.139,179.759,5.806,149.104
C04939=1177.961,-23.717,-44.153,179.762,5.806,149.103
C04940=1177.956,-23.447,-44.167,179.765,5.807,149.102
C04941=1177.949,-23.178,-44.181,179.767,5.807,149.102
C04942=1177.944,-22.927,-44.193,179.770,5.808,149.101
C04943=1177.939,-22.678,-44.206,179.772,5.808,149.101
C04944=1177.934,-22.428,-44.218,179.774,5.809,149.100
C04945=1177.929,-22.179,-44.231,179.777,5.810,149.099
C04946=1177.924,-21.930,-44.244,179.780,5.810,149.099
C04947=1177.919,-21.680,-44.257,179.782,5.811,149.098
C04948=1177.914,-21.430,-44.270,179.784,5.810,149.098
C04949=1177.908,-21.180,-44.282,179.787,5.811,149.097
C04950=1177.903,-20.931,-44.294,179.789,5.811,149.096
C04951=1177.899,-20.681,-44.307,179.791,5.812,149.096
C04952=1177.893,-20.432,-44.320,179.794,5.813,149.095
C04953=1177.888,-20.182,-44.333,179.797,5.813,149.094
C04954=1177.882,-19.933,-44.346,179.799,5.814,149.094
C04955=1177.878,-19.683,-44.359,179.802,5.814,149.093
C04956=1177.873,-19.433,-44.371,179.804,5.815,149.092
C04957=1177.868,-19.184,-44.384,179.806,5.815,149.092
C04958=1177.862,-18.934,-44.397,179.809,5.815,149.091
C04959=1177.857,-18.684,-44.409,179.811,5.816,149.091
C04960=1177.852,-18.434,-44.422,179.813,5.817,149.090
C04961=1177.847,-18.185,-44.434,179.816,5.817,149.089
C04962=1177.841,-17.935,-44.448,179.819,5.817,149.089
C04963=1177.836,-17.685,-44.461,179.821,5.818,149.088
C04964=1177.831,-17.436,-44.473,179.824,5.819,149.088
C04965=1177.827,-17.186,-44.486,179.826,5.819,149.087
C04966=1177.821,-16.936,-44.499,179.828,5.820,149.086
C04967=1177.816,-16.687,-44.512,179.831,5.821,149.086
C04968=1177.811,-16.438,-44.525,179.833,5.820,149.085
C04969=1177.805,-16.187,-44.538,179.835,5.821,149.085
C04970=1177.800,-15.938,-44.551,179.838,5.821,149.084
C04971=1177.795,-15.689,-44.563,179.841,5.822,149.083
C04972=1177.791,-15.439,-44.577,179.843,5.823,149.083
C04973=1177.785,-15.190,-44.590,179.845,5.823,149.082
C04974=1177.780,-14.941,-44.603,179.848,5.824,149.081
C04975=1177.775,-14.691,-44.616,179.850,5.824,149.081
C04976=1177.769,-14.441,-44.629,179.853,5.825,149.080
C04977=1177.764,-14.192,-44.642,179.856,5.825,149.079
C04978=1177.760,-13.942,-44.655,179.858,5.826,149.079
C04979=1177.754,-13.692,-44.668,179.860,5.827,149.078
C04980=1177.749,-13.442,-44.681,179.863,5.827,149.078
C04981=1177.744,-13.193,-44.693,179.865,5.827,149.077
C04982=1177.739,-12.944,-44.707,179.867,5.828,149.076
C04983=1177.734,-12.694,-44.720,179.870,5.828,149.076
C04984=1177.728,-12.444,-44.733,179.873,5.829,149.075
C04985=1177.723,-12.195,-44.746,179.875,5.829,149.075
C04986=1177.719,-11.945,-44.759,179.877,5.830,149.074
C04987=1177.713,-11.695,-44.772,179.880,5.830,149.073
C04988=1177.708,-11.445,-44.785,179.882,5.831,149.073
C04989=1177.704,-11.196,-44.798,179.885,5.832,149.072
C04990=1177.698,-10.947,-44.812,179.888,5.832,149.071
C04991=1177.693,-10.697,-44.825,179.890,5.833,149.071
C04992=1177.687,-10.447,-44.838,179.892,5.833,149.070
C04993=1177.683,-10.198,-44.851,179.895,5.834,149.070
C04994=1177.677,-9.948,-44.865,179.897,5.835,149.069
C04995=1177.672,-9.699,-44.877,179.900,5.835,149.068
C04996=1177.668,-9.449,-44.890,179.903,5.836,149.068
C04997=1177.662,-9.199,-44.903,179.905,5.836,149.067
C04998=1177.657,-8.950,-44.917,179.907,5.836,149.067
C04999=1177.652,-8.700,-44.930,179.909,5.836,149.066
C05000=1177.647,-8.450,-44.943,179.912,5.837,149.065
C05001=1177.642,-8.201,-44.957,179.914,5.838,149.065
C05002=1177.637,-7.951,-44.970,179.917,5.838,149.064
C05003=1177.631,-7.701,-44.983,179.919,5.839,149.064
C05004=1177.626,-7.452,-44.996,179.922,5.840,149.063
C05005=1177.621,-7.202,-45.010,179.924,5.840,149.062
C05006=1177.616,-6.953,-45.023,179.927,5.841,149.062
C05007=1177.611,-6.703,-45.036,179.929,5.841,149.061
C05008=1177.606,-6.454,-45.050,179.932,5.842,149.060
C05009=1177.601,-6.204,-45.063,179.934,5.843,149.060
C05010=1177.596,-5.955,-45.077,179.937,5.843,149.059
C05011=1177.591,-5.705,-45.090,179.939,5.843,149.058
C05012=1177.585,-5.455,-45.103,179.942,5.844,149.058
C05013=1177.580,-5.205,-45.117,179.944,5.845,149.057
C05014=1177.575,-4.956,-45.130,179.947,5.845,149.057
C05015=1177.570,-4.706,-45.143,179.949,5.846,149.056
C05016=1177.565,-4.457,-45.157,179.952,5.847,149.055
C05017=1177.560,-4.207,-45.170,179.954,5.847,149.055
C05018=1177.555,-3.958,-45.183,179.957,5.847,149.054
C05019=1177.550,-3.708,-45.197,179.959,5.848,149.054
C05020=1177.544,-3.459,-45.211,179.962,5.849,149.053
C05021=1177.540,-3.209,-45.224,179.965,5.849,149.052
C05022=1177.534,-2.959,-45.237,179.967,5.850,149.052
C05023=1177.530,-2.710,-45.251,179.969,5.851,149.051
C05024=1177.524,-2.460,-45.264,179.972,5.851,149.050
C05025=1177.519,-2.210,-45.278,179.974,5.852,149.050
C05026=1177.514,-1.961,-45.291,179.977,5.852,149.049
C05027=1177.509,-1.711,-45.305,179.979,5.853,149.049
C05028=1177.504,-1.462,-45.318,179.982,5.854,149.048
C05029=1177.499,-1.212,-45.332,179.984,5.854,149.047
C05030=1177.494,-0.962,-45.346,179.987,5.855,149.047
C05031=1177.489,-0.713,-45.359,179.989,5.855,149.046
C05032=1177.483,-0.463,-45.372,179.992,5.856,149.046
C05033=1177.478,-0.214,-45.386,179.994,5.856,149.045
C05034=1177.474,0.035,-45.400,179.997,5.857,149.044
C05035=1177.468,0.285,-45.413,179.999,5.858,149.044
C05036=1177.463,0.535,-45.427,-179.998,5.858,149.043
C05037=1177.458,0.784,-45.440,-179.996,5.859,149.043
C05038=1177.453,1.034,-45.454,-179.993,5.859,149.042
C05039=1177.448,1.284,-45.468,-179.991,5.860,149.041
C05040=1177.443,1.533,-45.481,-179.988,5.861,149.041
C05041=1177.438,1.783,-45.495,-179.986,5.861,149.040
C05042=1177.432,2.052,-45.510,-179.983,5.862,149.039
C05043=1177.426,2.321,-45.525,-179.980,5.862,149.039
C05044=1177.421,2.591,-45.539,-179.978,5.863,149.038
C05045=1177.415,2.860,-45.554,-179.976,5.863,149.038
C05046=1177.411,3.110,-45.568,-179.973,5.864,149.037
C05047=1177.405,3.359,-45.582,-179.970,5.864,149.036
C05048=1177.400,3.609,-45.596,-179.968,5.865,149.036
C05049=1177.395,3.858,-45.609,-179.966,5.866,149.035
C05050=1177.390,4.107,-45.623,-179.963,5.866,149.034
C05051=1177.385,4.358,-45.637,-179.961,5.867,149.034
C05052=1177.379,4.607,-45.651,-179.958,5.867,149.033
C05053=1177.375,4.856,-45.665,-179.955,5.868,149.032
C05054=1177.370,5.106,-45.679,-179.953,5.869,149.032
C05055=1177.364,5.355,-45.692,-179.951,5.869,149.031
C05056=1177.359,5.605,-45.706,-179.947,5.871,149.031
C05057=1177.355,5.855,-45.720,-179.945,5.871,149.030
C05058=1177.349,6.104,-45.734,-179.943,5.872,149.029
C05059=1177.344,6.354,-45.747,-179.940,5.872,149.029
C05060=1177.340,6.603,-45.761,-179.938,5.873,149.028
C05061=1177.334,6.852,-45.775,-179.935,5.874,149.028
C05062=1177.329,7.102,-45.790,-179.932,5.874,149.027
C05063=1177.324,7.352,-45.804,-179.930,5.875,149.027
C05064=1177.318,7.602,-45.817,-179.928,5.875,149.026
C05065=1177.314,7.851,-45.831,-179.925,5.876,149.025
C05066=1177.309,8.101,-45.845,-179.923,5.877,149.025
C05067=1177.303,8.350,-45.859,-179.920,5.877,149.024
C05068=1177.299,8.599,-45.873,-179.917,5.878,149.023
C05069=1177.293,8.850,-45.887,-179.915,5.879,149.023
C05070=1177.288,9.099,-45.901,-179.913,5.879,149.022
C05071=1177.283,9.348,-45.915,-179.910,5.879,149.021
C05072=1177.279,9.598,-45.929,-179.908,5.880,149.021
C05073=1177.274,9.848,-45.943,-179.905,5.881,149.020
C05074=1177.268,10.097,-45.957,-179.903,5.881,149.020
C05075=1177.263,10.346,-45.971,-179.900,5.882,149.019
C05076=1177.258,10.596,-45.985,-179.898,5.883,149.018
C05077=1177.253,10.846,-46.000,-179.895,5.883,149.018
C05078=1177.248,11.095,-46.014,-179.893,5.884,149.017
C05079=1177.242,11.345,-46.027,-179.890,5.885,149.017
C05080=1177.237,11.595,-46.041,-179.887,5.886,149.016
C05081=1177.232,11.844,-46.056,-179.885,5.887,149.016
C05082=1177.227,12.093,-46.070,-179.882,5.887,149.015
C05083=1177.222,12.343,-46.084,-179.880,5.887,149.014
C05084=1177.217,12.593,-46.098,-179.877,5.888,149.014
C05085=1177.212,12.843,-46.112,-179.875,5.889,149.013
C05086=1177.207,13.091,-46.126,-179.872,5.889,149.012
C05087=1177.202,13.341,-46.140,-179.870,5.890,149.012
C05088=1177.197,13.591,-46.154,-179.867,5.891,149.011
C05089=1177.192,13.840,-46.169,-179.865,5.891,149.011
C05090=1177.187,14.090,-46.183,-179.862,5.892,149.010
C05091=1177.182,14.339,-46.197,-179.860,5.892,149.009
C05092=1177.177,14.589,-46.211,-179.858,5.893,149.009
C05093=1177.172,14.839,-46.225,-179.854,5.895,149.008
C05094=1177.167,15.088,-46.240,-179.852,5.895,149.008
C05095=1177.162,15.337,-46.255,-179.850,5.896,149.007
C05096=1177.156,15.587,-46.269,-179.847,5.896,149.006
C05097=1177.151,15.836,-46.283,-179.844,5.897,149.006
C05098=1177.146,16.086,-46.298,-179.842,5.898,149.005
C05099=1177.141,16.336,-46.312,-179.839,5.898,149.005
C05100=1177.136,16.586,-46.326,-179.837,5.899,149.004
C05101=1177.131,16.835,-46.340,-179.835,5.900,149.003
C05102=1177.126,17.084,-46.354,-179.832,5.900,149.003
C05103=1177.121,17.334,-46.369,-179.829,5.900,149.002
C05104=1177.116,17.583,-46.384,-179.827,5.901,149.002
C05105=1177.111,17.833,-46.398,-179.824,5.903,149.001
C05106=1177.106,18.082,-46.412,-179.821,5.903,149.000
C05107=1177.101,18.332,-46.427,-179.819,5.904,149.000
C05108=1177.096,18.581,-46.440,-179.816,5.904,148.999
C05109=1177.091,18.831,-46.455,-179.814,5.905,148.999
C05110=1177.085,19.080,-46.470,-179.812,5.906,148.998
C05111=1177.080,19.330,-46.485,-179.809,5.906,148.997
C05112=1177.075,19.580,-46.499,-179.807,5.907,148.997
C05113=1177.070,19.829,-46.513,-179.804,5.908,148.996
C05114=1177.065,20.079,-46.527,-179.802,5.908,148.995
C05115=1177.061,20.328,-46.542,-179.799,5.910,148.995
C05116=1177.055,20.577,-46.556,-179.796,5.910,148.994
C05117=1177.050,20.827,-46.571,-179.793,5.911,148.994
C05118=1177.045,21.077,-46.585,-179.791,5.912,148.993
C05119=1177.040,21.326,-46.600,-179.789,5.912,148.993
C05120=1177.035,21.576,-46.615,-179.787,5.913,148.992
C05121=1177.030,21.825,-46.629,-179.784,5.913,148.991
C05122=1177.025,22.075,-46.644,-179.781,5.914,148.991
C05123=1177.020,22.325,-46.659,-179.778,5.916,148.990
C05124=1177.015,22.574,-46.673,-179.776,5.916,148.990
C05125=1177.010,22.823,-46.688,-179.773,5.916,148.989
C05126=1177.005,23.073,-46.702,-179.771,5.917,148.988
C05127=1177.000,23.322,-46.716,-179.768,5.918,148.988
C05128=1176.994,23.572,-46.732,-179.766,5.918,148.987
C05129=1176.989,23.821,-46.746,-179.764,5.919,148.987
C05130=1176.984,24.071,-46.761,-179.761,5.920,148.986
C05131=1176.980,24.320,-46.775,-179.758,5.921,148.986
C05132=1176.974,24.570,-46.790,-179.756,5.922,148.985
C05133=1176.969,24.820,-46.805,-179.753,5.922,148.984
C05134=1176.964,25.069,-46.820,-179.751,5.923,148.984
C05135=1176.959,25.319,-46.834,-179.748,5.924,148.983
C05136=1176.954,25.568,-46.850,-179.745,5.924,148.982
C05137=1176.949,25.818,-46.864,-179.743,5.925,148.982
C05138=1176.944,26.067,-46.879,-179.741,5.925,148.981
C05139=1176.939,26.316,-46.893,-179.737,5.927,148.981
C05140=1176.934,26.567,-46.908,-179.735,5.928,148.980
C05141=1176.929,26.816,-46.923,-179.733,5.928,148.979
C05142=1176.924,27.065,-46.937,-179.730,5.929,148.979
C05143=1176.919,27.315,-46.953,-179.728,5.929,148.978
C05144=1176.914,27.564,-46.967,-179.725,5.930,148.978
C05145=1176.909,27.814,-46.982,-179.722,5.932,148.977
C05146=1176.903,28.083,-46.998,-179.720,5.932,148.976
C05147=1176.898,28.351,-47.014,-179.717,5.933,148.976
C05148=1176.892,28.621,-47.030,-179.714,5.933,148.975
C05149=1176.887,28.889,-47.046,-179.711,5.934,148.974
C05150=1176.883,29.138,-47.061,-179.709,5.935,148.974
C05151=1176.877,29.388,-47.076,-179.706,5.936,148.973
C05152=1176.872,29.637,-47.091,-179.704,5.936,148.973
C05153=1176.867,29.887,-47.105,-179.702,5.937,148.972
C05154=1176.862,30.137,-47.121,-179.698,5.938,148.972
C05155=1176.857,30.386,-47.136,-179.696,5.939,148.971
C05156=1176.852,30.636,-47.151,-179.694,5.940,148.970
C05157=1176.847,30.885,-47.166,-179.691,5.940,148.970
C05158=1176.842,31.135,-47.180,-179.689,5.941,148.969
C05159=1176.837,31.384,-47.196,-179.686,5.942,148.969
C05160=1176.832,31.633,-47.211,-179.683,5.943,148.968
C05161=1176.827,31.884,-47.226,-179.681,5.944,148.967
C05162=1176.822,32.133,-47.241,-179.678,5.944,148.967
C05163=1176.817,32.382,-47.256,-179.676,5.945,148.966
C05164=1176.812,32.632,-47.271,-179.673,5.946,148.966
C05165=1176.807,32.881,-47.286,-179.670,5.947,148.965
C05166=1176.802,33.130,-47.301,-179.668,5.948,148.965
C05167=1176.797,33.380,-47.315,-179.665,5.948,148.964
C05168=1176.791,33.630,-47.331,-179.663,5.949,148.963
C05169=1176.787,33.879,-47.346,-179.660,5.950,148.963
C05170=1176.781,34.128,-47.362,-179.658,5.950,148.962
C05171=1176.776,34.378,-47.376,-179.655,5.952,148.962
C05172=1176.772,34.628,-47.392,-179.652,5.952,148.961
C05173=1176.767,34.877,-47.407,-179.650,5.953,148.960
C05174=1176.762,35.126,-47.422,-179.648,5.954,148.960
C05175=1176.757,35.376,-47.437,-179.645,5.954,148.959
C05176=1176.751,35.625,-47.452,-179.642,5.956,148.959
C05177=1176.747,35.875,-47.467,-179.640,5.956,148.958
C05178=1176.741,36.124,-47.483,-179.637,5.957,148.958
C05179=1176.737,36.374,-47.498,-179.635,5.958,148.957
C05180=1176.731,36.624,-47.513,-179.632,5.958,148.956
C05181=1176.727,36.873,-47.528,-179.629,5.960,148.956
C05182=1176.721,37.122,-47.544,-179.627,5.960,148.955
C05183=1176.716,37.372,-47.559,-179.624,5.961,148.954
C05184=1176.711,37.621,-47.574,-179.622,5.962,148.954
C05185=1176.706,37.871,-47.589,-179.619,5.962,148.953
C05186=1176.702,38.121,-47.605,-179.617,5.964,148.953
C05187=1176.696,38.370,-47.620,-179.614,5.964,148.952
C05188=1176.691,38.619,-47.636,-179.611,5.965,148.951
C05189=1176.686,38.868,-47.651,-179.609,5.966,148.951
C05190=1176.681,39.118,-47.666,-179.606,5.967,148.950
C05191=1176.677,39.368,-47.682,-179.604,5.968,148.950
C05192=1176.671,39.617,-47.697,-179.601,5.968,148.949
C05193=1176.666,39.866,-47.713,-179.598,5.969,148.949
C05194=1176.661,40.116,-47.727,-179.596,5.970,148.948
C05195=1176.656,40.366,-47.743,-179.593,5.971,148.947
C05196=1176.651,40.616,-47.759,-179.591,5.972,148.947
C05197=1176.646,40.865,-47.774,-179.588,5.972,148.946
C05198=1176.641,41.114,-47.789,-179.586,5.973,148.946
C05199=1176.636,41.363,-47.804,-179.583,5.975,148.945
C05200=1176.631,41.613,-47.820,-179.580,5.975,148.945
C05201=1176.626,41.863,-47.836,-179.578,5.976,148.944
C05202=1176.621,42.112,-47.851,-179.575,5.976,148.943
C05203=1176.616,42.361,-47.866,-179.573,5.977,148.943
C05204=1176.611,42.611,-47.882,-179.570,5.979,148.942
C05205=1176.606,42.861,-47.898,-179.567,5.979,148.942
C05206=1176.601,43.110,-47.913,-179.565,5.980,148.941
C05207=1176.596,43.359,-47.928,-179.563,5.980,148.941
C05208=1176.591,43.609,-47.944,-179.560,5.982,148.940
C05209=1176.587,43.858,-47.960,-179.557,5.983,148.939
C05210=1176.581,44.107,-47.976,-179.555,5.983,148.939
C05211=1176.576,44.357,-47.991,-179.552,5.984,148.938
C05212=1176.571,44.607,-48.007,-179.549,5.985,148.938
C05213=1176.566,44.856,-48.022,-179.547,5.986,148.937
C05214=1176.561,45.105,-48.038,-179.544,5.987,148.937
C05215=1176.556,45.355,-48.054,-179.542,5.988,148.936
C05216=1176.551,45.605,-48.069,-179.539,5.989,148.935
C05217=1176.546,45.854,-48.084,-179.536,5.989,148.935
C05218=1176.541,46.103,-48.101,-179.534,5.990,148.934
C05219=1176.536,46.353,-48.117,-179.532,5.991,148.934
C05220=1176.531,46.602,-48.132,-179.529,5.992,148.933
C05221=1176.526,46.852,-48.148,-179.526,5.993,148.933
C05222=1176.522,47.101,-48.163,-179.524,5.993,148.932
C05223=1176.516,47.351,-48.179,-179.521,5.995,148.931
C05224=1176.511,47.600,-48.195,-179.518,5.996,148.931
C05225=1176.506,47.850,-48.211,-179.516,5.997,148.930
C05226=1176.501,48.099,-48.227,-179.513,5.997,148.930
C05227=1176.496,48.348,-48.242,-179.511,5.999,148.929
C05228=1176.492,48.598,-48.258,-179.508,5.999,148.929
C05229=1176.486,48.847,-48.274,-179.505,6.000,148.928
C05230=1176.481,49.096,-48.289,-179.503,6.001,148.927
C05231=1176.476,49.347,-48.305,-179.500,6.002,148.927
C05232=1176.471,49.595,-48.322,-179.498,6.003,148.926
C05233=1176.466,49.845,-48.338,-179.495,6.003,148.926
C05234=1176.461,50.095,-48.353,-179.492,6.005,148.925
C05235=1176.457,50.343,-48.369,-179.490,6.005,148.925
C05236=1176.452,50.593,-48.385,-179.487,6.006,148.924
C05237=1176.446,50.843,-48.400,-179.485,6.007,148.923
C05238=1176.442,51.093,-48.416,-179.482,6.008,148.923
C05239=1176.437,51.342,-48.433,-179.480,6.009,148.922
C05240=1176.431,51.591,-48.448,-179.477,6.010,148.922
C05241=1176.427,51.841,-48.465,-179.474,6.011,148.921
C05242=1176.421,52.090,-48.481,-179.472,6.012,148.921
C05243=1176.417,52.340,-48.497,-179.469,6.013,148.920
C05244=1176.412,52.589,-48.513,-179.467,6.013,148.919
C05245=1176.406,52.838,-48.528,-179.464,6.014,148.919
C05246=1176.401,53.088,-48.544,-179.461,6.015,148.918
C05247=1176.396,53.337,-48.561,-179.459,6.016,148.918
C05248=1176.391,53.587,-48.577,-179.456,6.018,148.917
C05249=1176.386,53.836,-48.593,-179.453,6.018,148.917
C05250=1176.381,54.104,-48.610,-179.451,6.019,148.916
C05251=1176.376,54.374,-48.627,-179.448,6.020,148.915
C05252=1176.370,54.642,-48.644,-179.445,6.021,148.915
C05253=1176.365,54.910,-48.662,-179.442,6.022,148.914
C05254=1176.360,55.160,-48.678,-179.440,6.023,148.914
C05255=1176.355,55.409,-48.694,-179.437,6.024,148.913
C05256=1176.350,55.659,-48.710,-179.435,6.025,148.913
C05257=1176.345,55.908,-48.727,-179.432,6.026,148.912
C05258=1176.341,56.158,-48.743,-179.429,6.027,148.911
C05259=1176.335,56.407,-48.759,-179.427,6.028,148.911
C05260=1176.331,56.657,-48.775,-179.424,6.028,148.910
C05261=1176.326,56.906,-48.791,-179.422,6.029,148.910
C05262=1176.320,57.155,-48.807,-179.419,6.031,148.909
C05263=1176.316,57.404,-48.823,-179.417,6.031,148.909
C05264=1176.310,57.654,-48.839,-179.414,6.032,148.908
C05265=1176.306,57.903,-48.856,-179.411,6.034,148.907
C05266=1176.301,58.153,-48.872,-179.409,6.034,148.907
C05267=1176.295,58.403,-48.888,-179.406,6.035,148.906
C05268=1176.291,58.652,-48.905,-179.403,6.036,148.906
C05269=1176.285,58.901,-48.921,-179.401,6.037,148.905
C05270=1176.281,59.151,-48.937,-179.398,6.038,148.905
C05271=1176.276,59.400,-48.954,-179.395,6.039,148.904
C05272=1176.271,59.650,-48.970,-179.393,6.040,148.904
C05273=1176.266,59.899,-48.986,-179.390,6.041,148.903
C05274=1176.261,60.148,-49.003,-179.388,6.042,148.902
C05275=1176.255,60.398,-49.019,-179.385,6.043,148.902
C05276=1176.251,60.647,-49.035,-179.382,6.044,148.901
C05277=1176.246,60.896,-49.052,-179.380,6.045,148.901
C05278=1176.241,61.146,-49.068,-179.377,6.046,148.900
C05279=1176.237,61.396,-49.084,-179.374,6.047,148.900
C05280=1176.231,61.644,-49.101,-179.372,6.048,148.899
C05281=1176.226,61.894,-49.118,-179.369,6.048,148.898
C05282=1176.221,62.144,-49.134,-179.367,6.050,148.898
C05283=1176.216,62.393,-49.150,-179.364,6.051,148.897
C05284=1176.211,62.642,-49.167,-179.361,6.051,148.897
C05285=1176.207,62.891,-49.183,-179.359,6.053,148.896
C05286=1176.201,63.142,-49.200,-179.356,6.053,148.896
C05287=1176.196,63.391,-49.216,-179.354,6.054,148.895
C05288=1176.192,63.640,-49.233,-179.351,6.056,148.895
C05289=1176.187,63.889,-49.249,-179.349,6.057,148.894
C05290=1176.182,64.138,-49.266,-179.345,6.058,148.893
C05291=1176.177,64.389,-49.282,-179.343,6.059,148.893
C05292=1176.172,64.637,-49.299,-179.341,6.059,148.892
C05293=1176.167,64.887,-49.315,-179.338,6.061,148.892
C05294=1176.163,65.136,-49.332,-179.335,6.061,148.891
C05295=1176.157,65.386,-49.349,-179.333,6.062,148.891
C05296=1176.152,65.635,-49.365,-179.330,6.064,148.890
C05297=1176.147,65.884,-49.382,-179.328,6.065,148.890
C05298=1176.142,66.134,-49.398,-179.325,6.066,148.889
C05299=1176.137,66.384,-49.415,-179.322,6.067,148.889
C05300=1176.132,66.632,-49.431,-179.320,6.067,148.888
C05301=1176.127,66.882,-49.449,-179.317,6.069,148.888
C05302=1176.122,67.132,-49.465,-179.314,6.069,148.887
C05303=1176.117,67.381,-49.482,-179.312,6.071,148.886
C05304=1176.113,67.630,-49.498,-179.309,6.072,148.886
C05305=1176.108,67.880,-49.515,-179.307,6.073,148.885
C05306=1176.103,68.129,-49.532,-179.304,6.074,148.885
C05307=1176.097,68.378,-49.549,-179.302,6.075,148.884
C05308=1176.093,68.628,-49.566,-179.299,6.075,148.884
C05309=1176.088,68.877,-49.582,-179.296,6.077,148.883
C05310=1176.083,69.126,-49.599,-179.294,6.078,148.882
C05311=1176.078,69.376,-49.616,-179.291,6.079,148.882
C05312=1176.074,69.625,-49.633,-179.288,6.080,148.881
C05313=1176.068,69.875,-49.649,-179.286,6.081,148.881
C05314=1176.063,70.124,-49.666,-179.283,6.082,148.880
C05315=1176.058,70.374,-49.683,-179.281,6.083,148.880
C05316=1176.054,70.623,-49.700,-179.277,6.084,148.879
C05317=1176.049,70.872,-49.716,-179.275,6.085,148.879
C05318=1176.043,71.122,-49.734,-179.272,6.086,148.878
C05319=1176.039,71.371,-49.750,-179.270,6.087,148.878
C05320=1176.033,71.620,-49.767,-179.267,6.088,148.877
C05321=1176.029,71.869,-49.785,-179.265,6.090,148.877
C05322=1176.024,72.119,-49.802,-179.262,6.090,148.876
C05323=1176.019,72.369,-49.819,-179.259,6.092,148.876
C05324=1176.013,72.618,-49.835,-179.257,6.092,148.875
C05325=1176.009,72.867,-49.852,-179.254,6.093,148.874
C05326=1176.004,73.117,-49.869,-179.251,6.095,148.874
C05327=1175.999,73.366,-49.886,-179.249,6.095,148.873
C05328=1175.995,73.615,-49.903,-179.246,6.097,148.873
C05329=1175.989,73.864,-49.920,-179.244,6.098,148.872
C05330=1175.985,74.114,-49.937,-179.241,6.099,148.872
C05331=1175.979,74.364,-49.954,-179.238,6.100,148.871
C05332=1175.975,74.613,-49.971,-179.236,6.100,148.871
C05333=1175.970,74.862,-49.989,-179.233,6.102,148.870
C05334=1175.964,75.111,-50.006,-179.230,6.103,148.869
C05335=1175.960,75.361,-50.022,-179.228,6.104,148.869
C05336=1175.955,75.611,-50.040,-179.225,6.105,148.868
C05337=1175.950,75.860,-50.057,-179.222,6.107,148.868
C05338=1175.945,76.109,-50.074,-179.220,6.107,148.867
C05339=1175.940,76.358,-50.091,-179.217,6.109,148.867
C05340=1175.935,76.608,-50.108,-179.215,6.110,148.866
C05341=1175.931,76.857,-50.125,-179.212,6.110,148.866
C05342=1175.925,77.107,-50.143,-179.209,6.112,148.865
C05343=1175.920,77.356,-50.160,-179.207,6.112,148.865
C05344=1175.916,77.605,-50.177,-179.204,6.114,148.864
C05345=1175.910,77.854,-50.194,-179.201,6.115,148.864
C05346=1175.906,78.104,-50.211,-179.199,6.116,148.863
C05347=1175.901,78.353,-50.229,-179.196,6.117,148.863
C05348=1175.896,78.603,-50.246,-179.193,6.119,148.862
C05349=1175.891,78.852,-50.263,-179.191,6.119,148.861
C05350=1175.886,79.102,-50.281,-179.188,6.121,148.861
C05351=1175.881,79.351,-50.298,-179.185,6.121,148.860
C05352=1175.876,79.599,-50.315,-179.183,6.123,148.860
C05353=1175.871,79.849,-50.332,-179.181,6.124,148.859
C05354=1175.866,80.118,-50.351,-179.177,6.125,148.859
C05355=1175.861,80.386,-50.370,-179.175,6.126,148.858
C05356=1175.855,80.654,-50.388,-179.172,6.128,148.858
C05357=1175.850,80.923,-50.407,-179.169,6.129,148.857
C05358=1175.845,81.172,-50.425,-179.167,6.130,148.857
C05359=1175.841,81.422,-50.441,-179.163,6.131,148.856
C05360=1175.836,81.671,-50.459,-179.161,6.132,148.856
C05361=1175.830,81.921,-50.477,-179.158,6.133,148.855
C05362=1175.825,82.170,-50.495,-179.156,6.134,148.855
C05363=1175.821,82.419,-50.511,-179.153,6.136,148.854
C05364=1175.816,82.669,-50.529,-179.151,6.136,148.853
C05365=1175.811,82.918,-50.547,-179.147,6.138,148.853
C05366=1175.806,83.167,-50.564,-179.145,6.139,148.852
C05367=1175.801,83.416,-50.581,-179.143,6.140,148.852
C05368=1175.796,83.666,-50.599,-179.140,6.141,148.851
C05369=1175.791,83.915,-50.616,-179.138,6.142,148.851
C05370=1175.786,84.164,-50.634,-179.135,6.143,148.850
C05371=1175.782,84.413,-50.651,-179.132,6.144,148.850
C05372=1175.776,84.663,-50.669,-179.129,6.145,148.849
C05373=1175.772,84.912,-50.687,-179.127,6.146,148.849
C05374=1175.766,85.162,-50.704,-179.124,6.148,148.848
C05375=1175.762,85.411,-50.721,-179.122,6.149,148.848
C05376=1175.757,85.660,-50.739,-179.119,6.150,148.847
C05377=1175.752,85.910,-50.757,-179.116,6.152,148.847
C05378=1175.747,86.159,-50.775,-179.114,6.153,148.846
C05379=1175.742,86.408,-50.793,-179.110,6.154,148.846
C05380=1175.737,86.658,-50.810,-179.108,6.155,148.845
C05381=1175.733,86.907,-50.827,-179.105,6.156,148.844
C05382=1175.728,87.156,-50.845,-179.103,6.157,148.844
C05383=1175.723,87.406,-50.862,-179.100,6.159,148.844
C05384=1175.718,87.655,-50.880,-179.098,6.159,148.843
C05385=1175.713,87.904,-50.898,-179.095,6.161,148.843
C05386=1175.708,88.153,-50.916,-179.092,6.162,148.842
C05387=1175.703,88.403,-50.934,-179.089,6.163,148.841
C05388=1175.698,88.652,-50.952,-179.087,6.164,148.841
C05389=1175.694,88.901,-50.969,-179.084,6.165,148.840
C05390=1175.689,89.150,-50.987,-179.082,6.166,148.840
C05391=1175.684,89.400,-51.004,-179.079,6.168,148.839
C05392=1175.679,89.650,-51.023,-179.077,6.169,148.839
C05393=1175.674,89.899,-51.041,-179.073,6.170,148.838
C05394=1175.669,90.148,-51.059,-179.071,6.171,148.838
C05395=1175.664,90.398,-51.077,-179.069,6.173,148.837
C05396=1175.660,90.647,-51.095,-179.066,6.173,148.837
C05397=1175.654,90.897,-51.112,-179.063,6.175,148.836
C05398=1175.649,91.146,-51.130,-179.060,6.176,148.836
C05399=1175.645,91.395,-51.148,-179.058,6.177,148.835
C05400=1175.640,91.644,-51.166,-179.055,6.179,148.835
C05401=1175.635,91.893,-51.184,-179.053,6.179,148.834
C05402=1175.630,92.143,-51.202,-179.050,6.181,148.834
C05403=1175.625,92.392,-51.220,-179.047,6.182,148.833
C05404=1175.621,92.642,-51.238,-179.045,6.183,148.833
C05405=1175.616,92.891,-51.256,-179.042,6.184,148.832
C05406=1175.610,93.141,-51.273,-179.039,6.186,148.832
C05407=1175.606,93.390,-51.291,-179.037,6.186,148.831
C05408=1175.601,93.639,-51.309,-179.034,6.188,148.831
C05409=1175.596,93.888,-51.327,-179.031,6.190,148.830
C05410=1175.591,94.137,-51.345,-179.029,6.190,148.830
C05411=1175.586,94.386,-51.363,-179.026,6.192,148.829
C05412=1175.582,94.636,-51.382,-179.024,6.193,148.829
C05413=1175.577,94.885,-51.399,-179.020,6.194,148.828
C05414=1175.572,95.135,-51.417,-179.018,6.195,148.828
C05415=1175.567,95.384,-51.435,-179.016,6.197,148.827
C05416=1175.562,95.633,-51.453,-179.012,6.198,148.827
C05417=1175.556,95.882,-51.472,-179.010,6.199,148.826
C05418=1175.552,96.132,-51.490,-179.008,6.201,148.826
C05419=1175.547,96.382,-51.508,-179.005,6.201,148.825
C05420=1175.542,96.630,-51.527,-179.002,6.203,148.825
C05421=1175.538,96.879,-51.545,-179.000,6.203,148.824
C05422=1175.533,97.128,-51.563,-178.997,6.205,148.824
C05423=1175.528,97.378,-51.581,-178.994,6.207,148.823
C05424=1175.523,97.627,-51.599,-178.992,6.207,148.823
C05425=1175.518,97.877,-51.618,-178.989,6.209,148.822
C05426=1175.513,98.126,-51.636,-178.987,6.210,148.822
C05427=1175.508,98.375,-51.654,-178.983,6.211,148.821
C05428=1175.503,98.625,-51.672,-178.981,6.213,148.821
C05429=1175.499,98.874,-51.691,-178.978,6.214,148.820
C05430=1175.494,99.123,-51.709,-178.975,6.215,148.820
C05431=1175.488,99.372,-51.727,-178.973,6.216,148.819
C05432=1175.484,99.622,-51.745,-178.970,6.218,148.819
C05433=1175.479,99.871,-51.764,-178.967,6.219,148.818
C05434=1175.475,100.120,-51.782,-178.965,6.220,148.818
C05435=1175.470,100.369,-51.800,-178.962,6.222,148.817
C05436=1175.464,100.619,-51.819,-178.960,6.223,148.817
C05437=1175.460,100.869,-51.837,-178.957,6.224,148.816
C05438=1175.455,101.117,-51.856,-178.954,6.226,148.816
C05439=1175.450,101.366,-51.874,-178.952,6.227,148.815
C05440=1175.445,101.616,-51.893,-178.949,6.228,148.815
C05441=1175.440,101.866,-51.911,-178.947,6.229,148.814
C05442=1175.436,102.114,-51.930,-178.944,6.231,148.814
C05443=1175.431,102.363,-51.948,-178.941,6.232,148.813
C05444=1175.425,102.613,-51.966,-178.938,6.233,148.813
C05445=1175.421,102.862,-51.985,-178.936,6.235,148.812
C05446=1175.416,103.111,-52.003,-178.933,6.235,148.812
C05447=1175.411,103.360,-52.021,-178.930,6.237,148.811
C05448=1175.406,103.610,-52.041,-178.928,6.239,148.811
C05449=1175.402,103.859,-52.059,-178.925,6.239,148.810
C05450=1175.397,104.108,-52.077,-178.922,6.241,148.810
C05451=1175.392,104.358,-52.097,-178.920,6.243,148.809
C05452=1175.387,104.607,-52.114,-178.917,6.243,148.809
C05453=1175.382,104.856,-52.133,-178.914,6.245,148.808
C05454=1175.377,105.106,-52.152,-178.912,6.247,148.808
C05455=1175.372,105.355,-52.170,-178.909,6.247,148.807
C05456=1175.367,105.604,-52.189,-178.906,6.249,148.807
C05457=1175.363,105.854,-52.208,-178.904,6.250,148.806
C05458=1175.358,106.121,-52.228,-178.901,6.251,148.806
C05459=1175.352,106.390,-52.248,-178.898,6.253,148.805
C05460=1175.346,106.659,-52.268,-178.895,6.254,148.805
C05461=1175.342,106.927,-52.288,-178.892,6.256,148.804
C05462=1175.337,107.176,-52.307,-178.890,6.256,148.804
C05463=1175.332,107.425,-52.326,-178.887,6.258,148.803
C05464=1175.328,107.675,-52.344,-178.884,6.260,148.803
C05465=1175.322,107.924,-52.363,-178.882,6.260,148.802
C05466=1175.318,108.174,-52.382,-178.879,6.262,148.802
C05467=1175.313,108.422,-52.401,-178.876,6.264,148.801
C05468=1175.308,108.672,-52.419,-178.874,6.264,148.801
C05469=1175.303,108.921,-52.439,-178.871,6.266,148.800
C05470=1175.298,109.170,-52.457,-178.868,6.268,148.800
C05471=1175.294,109.420,-52.476,-178.866,6.268,148.799
C05472=1175.289,109.668,-52.495,-178.863,6.270,148.799
C05473=1175.284,109.918,-52.513,-178.860,6.272,148.799
C05474=1175.279,110.167,-52.533,-178.858,6.273,148.798
C05475=1175.274,110.416,-52.551,-178.855,6.274,148.798
C05476=1175.269,110.666,-52.570,-178.852,6.276,148.797
C05477=1175.265,110.915,-52.589,-178.850,6.277,148.797
C05478=1175.260,111.164,-52.608,-178.847,6.278,148.796
C05479=1175.255,111.413,-52.626,-178.844,6.280,148.796
C05480=1175.250,111.663,-52.646,-178.842,6.281,148.795
C05481=1175.245,111.912,-52.665,-178.839,6.282,148.795
C05482=1175.240,112.161,-52.683,-178.836,6.284,148.794
C05483=1175.235,112.410,-52.703,-178.834,6.285,148.794
C05484=1175.231,112.659,-52.722,-178.831,6.287,148.793
C05485=1175.226,112.909,-52.741,-178.828,6.288,148.793
C05486=1175.221,113.158,-52.759,-178.825,6.290,148.792
C05487=1175.216,113.407,-52.779,-178.823,6.291,148.792
C05488=1175.211,113.656,-52.798,-178.820,6.292,148.791
C05489=1175.207,113.906,-52.817,-178.817,6.294,148.791
C05490=1175.201,114.155,-52.836,-178.815,6.295,148.791
C05491=1175.197,114.404,-52.855,-178.812,6.296,148.790
C05492=1175.192,114.653,-52.874,-178.809,6.298,148.789
C05493=1175.187,114.903,-52.894,-178.807,6.299,148.789
